ACTION FlowInit:
IF NOT station.xIniting THEN
  station.iStepInit:=0;    
ELSE
//--------------------------------------------初始化步序----------------------------------
CASE station.iStepInit OF	
 0://  
  	IF station.xIniting THEN	
  	  station.iStepInit:=10;	
  	END_IF	
10://复位数据
  station.iStepInit:=20;	
20://停止皮带线
		ATV12.xIMotorStop:=TRUE;
		 station.iStepInit:=999;	
999://初始化完成	
	station.iStepInit:=0;
	station.xInitDone:=TRUE;  
END_CASE
END_IF
END_ACTION

ACTION General:
{region "停止"}
tStopDelay(IN:= fbMachine[1].xManualMode, PT:=T#60S , Q=> , ET=> );
IF tStopDelay.Q THEN
		station.xRunningOffProhibit:=FALSE;
ELSIF  station.iStepAuto =10 THEN
		station.xRunningOffProhibit:=TRUE;
END_IF	 
{endregion}
END_ACTION

ACTION ILC:

//---------------------------------------------------工站可执行-------------------------------------------------------
station.xCanRun :=TRUE ;

//---------------------------------------------------气缸动作条件-------------------------------------------

//变频器
ATV12.xIDeviceRunning:=station.xSingleRunning;
END_ACTION

ACTION Z_Output:

END_ACTION

END_PROGRAM

// ---- POUs/003_FB/0006_ATV/FB_ATV12.TcPOU
FUNCTION_BLOCK FB_ATV12
(*
********************************************************************************
* Name: FB_Encoder
*
* Author:  AutomanH
* Version: 1.0.0
*
* Description:
*   Schneider ATV12 
* Remarks:
*
* Revisions:
* 
*********************************************************************************)
VAR_INPUT
 xIMotorStart:BOOL; //电机启动
 xIMotorStartHMI:BOOL;
 xIMotorStop:BOOL; //电机停止
 xIMotorStopHMI:BOOL;
 xIAutoMode:BOOL;
 xIManualMode:BOOL;
 xIEStop:BOOL;
 xIDeviceRunning:BOOL;
END_VAR
VAR_OUTPUT
 xQMotorStart:BOOL;//变频器电机启动
 arxQMotorSpeedCmd:ARRAY[1..2] OF BOOL;//预制速度
 xQRev:BOOL;//备用
END_VAR
VAR
 	MotorStartR_TRIG:R_TRIG;
	MotorStopR_TRIG:R_TRIG;
	MotorEStopR_TRIG:R_TRIG;
END_VAR

//变频器（2线 漏型）
MotorStartR_TRIG(CLK:=( xIManualMode AND   xIMotorStartHMI ) OR ( (xIAutoMode OR xIDeviceRunning ) AND   xIMotorStart) , Q=> );
MotorStopR_TRIG(CLK:= ( xIManualMode AND   xIMotorStopHMI ) OR ((xIAutoMode OR xIDeviceRunning ) AND xIMotorStop), Q=> );
MotorEStopR_TRIG(CLK:=xIEStop, Q=> );
IF  MotorStartR_TRIG.Q THEN
			xQMotorStart	:=TRUE;//	热缩封膜出料线体¶电机正转/停止
ELSIF	MotorStopR_TRIG.Q	 THEN
			xQMotorStart	:=FALSE;//	热缩封膜出料线体¶电机正转/停止
		
END_IF
	arxQMotorSpeedCmd[1]	:=FALSE;//	热缩封膜出料线体¶电机（预约速度20HZ)
	arxQMotorSpeedCmd[2]	:=TRUE;//	热缩封膜出料线体¶电机（预约速度50HZ）
	
	
	xQRev	:=FALSE;//	热缩封膜出料线体¶电机（未使用）
	
		xIMotorStopHMI:=FALSE;
		xIMotorStop:=FALSE;
		xIMotorStartHMI:=FALSE;
		xIMotorStart:=FALSE;

END_FUNCTION_BLOCK

// ---- POUs/001_Station/S13_Labeling.TcPOU
PROGRAM S13_Labeling
VAR
	//工站
	station					: REFERENCE TO FB_Station:=fbstation[13];
	//气缸
	fbHOZCyl_1			:REFERENCE TO FB_Cylinder:=fbCylinder[36];	//	分料气缸1
	//延时
	arTonDelay :ARRAY[1..20] OF TON;
	//返回值
	UdiReturnValue :ARRAY[1..20] OF UDINT;
	//贴标机
	xLabelJobRdySignal:BOOL;//	贴标机JOBRDY信号
	xLabelReadySignal:BOOL;//	贴标机READY信号
	xLabelErrorSignal:BOOL;//	贴标机ERROR信号
	i: INT;
	xQLabelStart: BOOL;			//	贴标机Start 
	xQLabelRibwarn: BOOL; //	贴标机RIBWARN
	xQLabelReset: BOOL;   //	贴标机RESET  
	
	xQLabelCompleted:BOOL;//贴标完成信号  给PC
	// 贴标到位传感器
	arSensorReached: ARRAY[1..2]of BOOL;
	
	// 设备停止延时
	tStopDelay: TON;
END_VAR

A_Input();
Alarm();
Delay();
FlowAuto();
FlowInit();
General();
ILC();
TipAuto();
TipManual();
Z_Output();

ACTION A_Input:
//气缸
fbHOZCyl_1.xWP_Sensor:=	IxS11HOZCylWP	;//	贴标处推料气缸¶动点
fbHOZCyl_1.xHP_Sensor:=	IxS11HOZCylHP	;//	贴标处推料气缸¶原点
//贴标机

xLabelJobRdySignal:=IxLabelJobRdySignal	;//	贴标机JOBRDY信号
xLabelReadySignal:=IxLabelReadySignal	;//	贴标机READY信号
xLabelErrorSignal:= NOT IxLabelErrorSignal	;//	贴标机ERROR信号

//贴标机到位传感器
arSensorReached[1]:=IxS11SensorReached1	;//	贴标工位¶检查到位传感器1
arSensorReached[2]:=IxS11SensorReached2;//	贴标工位¶检查到位传感器2
END_ACTION

ACTION Alarm:

station.adwAlarm[1].00:=station.xInitTimeout;	  			//S08Label 初始化超时
END_ACTION

ACTION Delay:
(*arTonDelay[01](IN:= , PT:=T#0.1S , Q=> , ET=> );*)//TipAuto使用
arTonDelay[02](IN:= station.iStepAuto=100 , PT:=T#1S , Q=> , ET=> );//贴标识用
arTonDelay[03](IN:=station.iStepAuto =40  , PT:=stData.TimeS[1] , Q=> , ET=> );//计算贴标延时
arTonDelay[04](IN:= , PT:=T#0.1S , Q=> , ET=> );
arTonDelay[05](IN:= , PT:=T#0.1S , Q=> , ET=> );
arTonDelay[06](IN:= , PT:=T#0.1S , Q=> , ET=> );
arTonDelay[07](IN:= , PT:=T#0.1S , Q=> , ET=> );
arTonDelay[08](IN:= , PT:=T#0.1S , Q=> , ET=> );
arTonDelay[09](IN:= , PT:=T#0.1S , Q=> , ET=> );
END_ACTION

ACTION FlowAuto:

//-----------------------------------------初始化是否完成判断----------------------------------------------
IF NOT station.xInitDone 
THEN
 	station.iStepAuto:=0;
 	station.xDone:=FALSE;
ELSIF station.xRunning  OR   station.xRunningOffProhibit
THEN
//-----------------------------------------动作步骤--------------------------------------------------------
CASE station.iStepAuto OF	  
	0: //----Home Step，等待启动----
		IF station.xDisabled 
			AND station.xCanRun 
			AND NOT fbMachine[1].xStopped 
			AND NOT station.xSingleRunning 
		THEN
			station.xDone:=TRUE;
		END_IF
		
		IF  station.xSingleRunning 
			OR station.xCanRun 
			AND NOT station.xDone 
			AND NOT station.xDisabled 
			AND NOT fbMachine[1].xStopped
		THEN
			station.xCycleEnable:=TRUE;
			station.xDone:= FALSE;  
			station.xRunningOffProhibit := TRUE ;//运行中信号Off禁止
			station.iStepAuto:= 10;
		END_IF
    10: //复位数据 
			xQLabelStart:=FALSE;			//	贴标机Start
			station.iStepAuto:=20;
		20://等待第一个传感器感应到
			IF  arSensorReached[1] THEN
						station.iStepAuto:=30;	
			END_IF
		30://等待两个传感器都感应到
				IF  arSensorReached[1]  AND arSensorReached[2] THEN
						station.iStepAuto:=40;	
			END_IF
		40://计算延时触发贴标
				IF   arTonDelay[03].Q THEN
					station.iStepAuto:=100;
				END_IF
		100://开始触发贴标
					xQLabelStart:=TRUE;			//	贴标机Start
					IF	arTonDelay[02].Q THEN
							station.iStepAuto:=110;
					END_IF							
		110://等待贴标完成
					xQLabelStart:=FALSE;			//	贴标机stop
					station.iStepAuto:=999;

		999://----Single Run Finish----
				station.iStepAuto :=0;
				IF NOT station.xSingleContinuousRun THEN
					station.xSingleRunFlag:=FALSE;
				END_IF
				
				station.xCycleEnable:=FALSE;	
				//station.xDone:=TRUE;
			//	station.xRunningOffProhibit := FALSE ;//运行中信号Off禁止
	ELSE
		;	
END_CASE



END_IF
END_ACTION

ACTION FlowInit:
IF NOT station.xIniting THEN
  station.iStepInit:=0;    
ELSE
//--------------------------------------------初始化步序----------------------------------
CASE station.iStepInit OF	
 0://  
  	IF station.xIniting THEN	
  	  station.iStepInit:=10;	
  	END_IF	
10://复位数据
    station.iStepInit:=999;	
		xQLabelStart:=FALSE;			//	贴标机Start
999://初始化完成	
	station.iStepInit:=0;
	station.xInitDone:=TRUE;  
END_CASE
END_IF
END_ACTION

ACTION General:
{region "停止"}
tStopDelay(IN:= fbMachine[1].xManualMode, PT:=T#60S , Q=> , ET=> );
IF tStopDelay.Q THEN
		station.xRunningOffProhibit:=FALSE;
ELSIF  station.iStepAuto =10 THEN
		station.xRunningOffProhibit:=TRUE;
END_IF	 
{endregion}
END_ACTION

ACTION ILC:

//---------------------------------------------------工站可执行-------------------------------------------------------
station.xCanRun :=TRUE ;

//---------------------------------------------------气缸动作条件-------------------------------------------
fbHOZCyl_1.xOffILC	:=	TRUE	;
fbHOZCyl_1.xOnILC	:=	TRUE; 


//---------------------------------------------------伺服动作条件-------------------------------------------
END_ACTION

ACTION TipAuto:

//------------------------------------------------AutoTip Cylinder--------------------------------

//------------------------------------------------AutoTip Servo--------------------------------
//**************************************
END_ACTION

ACTION TipManual:
//--------------------------------------------ManualTip------------------------------------------------------

//-------------------------------------------气缸提示---------------------------------------------------------




/////////////////////////////////////////////////////////////////////////////////////////////////////////////////
END_ACTION

ACTION Z_Output:
(**************************气缸输出********************************)
QxS11HOZCylWP	:=fbHOZCyl_1.xWP_Valve;//	贴标处推料气缸¶动点
QxS11HOZCylHP	:=fbHOZCyl_1.xHP_Valve;//	贴标处推料气缸¶原点
//贴标机
QxLabelStart	:=xQLabelStart;			//	贴标机Start
QxLabelRibwarn:=xQLabelRibwarn;	//	贴标机RIBWARN
QxLabelReset	:=xQLabelReset;		//	贴标机RESET
END_ACTION

END_PROGRAM

// ---- POUs/001_Station/S14_LabelChecking.TcPOU
PROGRAM S14_LabelChecking
VAR
	//工站
	station					: REFERENCE TO FB_Station:=fbstation[14];
	
//气缸
	fbHOZCyl_1			:REFERENCE TO FB_Cylinder:=fbCylinder[37];	//	推料气缸1
	fbHOZCyl_2			:REFERENCE TO FB_Cylinder:=fbCylinder[38];	//	推料气缸2
//相机
	Camera   : 	 REFERENCE TO FB_Camera:=fbCamera[18]; 
	
	//延时
	arTonDelay :ARRAY[1..20] OF TON;
	//返回值
	UdiReturnValue :ARRAY[1..20] OF UDINT;
	i: INT;
 //传感器
	arxBoxCheckSensor: ARRAY[1..2] OF BOOL;
	// //需要推到NG位置
	xNGFlag: BOOL;
	//运行结束
	XFlowAutoDone:BOOL;
		// 设备停止延时
	tStopDelay: TON;
END_VAR

A_Input();
Alarm();
Delay();
FlowAuto();
FlowInit();
General();
ILC();
TipAuto();
TipManual();
Z_Output();

ACTION A_Input:
//气缸
fbHOZCyl_1.xWP_Sensor:=					IxS12HOZCyl_1WP;//	贴标检测工位¶推料气缸1¶动点
fbHOZCyl_1.xHP_Sensor:=					IxS12HOZCyl_1HP;//	贴标检测工位¶推料气缸1¶原点
fbHOZCyl_2.xWP_Sensor:=					IxS12HOZCyl_2HP;//	贴标检测工位¶推料气缸2¶动点
fbHOZCyl_2.xHP_Sensor:=					IxS12HOZCyl_2WP;//	贴标检测工位W推料气缸2¶原点

//传感器
arxBoxCheckSensor[1] :=IxS12SensorReached;	//相机检测处
END_ACTION

ACTION Alarm:
//
station.adwAlarm[1].00:=station.xInitTimeout;	  			//S08Label 初始化超时
//station.adwAlarm[1].01:=TRUE;	  			//S14贴标工位相机检测超时，请检查
END_ACTION

ACTION Delay:
(*arTonDelay[01](IN:= , PT:=T#0.1S , Q=> , ET=> );*)//TipAuto使用
arTonDelay[02](IN:= 	station.iStepAuto=60 , PT:=T#1S , Q=> , ET=> );//已使用
arTonDelay[03](IN:=   , PT:=T#1S , Q=> , ET=> );
arTonDelay[04](IN:= , PT:=T#0.1S , Q=> , ET=> );
arTonDelay[05](IN:= , PT:=T#0.1S , Q=> , ET=> );
arTonDelay[06](IN:= , PT:=T#0.1S , Q=> , ET=> );
arTonDelay[07](IN:= , PT:=T#0.1S , Q=> , ET=> );
arTonDelay[08](IN:= , PT:=T#0.1S , Q=> , ET=> );
arTonDelay[09](IN:= , PT:=T#0.1S , Q=> , ET=> );
END_ACTION

ACTION FlowAuto:

//-----------------------------------------初始化是否完成判断----------------------------------------------
IF NOT station.xInitDone 
THEN
 	station.iStepAuto:=0;
 	station.xDone:=FALSE;
ELSIF station.xRunning  OR   station.xRunningOffProhibit
THEN
//-----------------------------------------动作步骤--------------------------------------------------------
CASE station.iStepAuto OF	  
	0: //----Home Step，等待启动----
		IF station.xDisabled 
			AND station.xCanRun 
			AND NOT fbMachine[1].xStopped 
			AND NOT station.xSingleRunning 
		THEN
			station.xDone:=TRUE;
		END_IF
		
		IF  station.xSingleRunning 
			OR station.xCanRun 
			AND NOT station.xDone 
			AND NOT station.xDisabled 
			AND NOT fbMachine[1].xStopped
		THEN
			station.xCycleEnable:=TRUE;
			station.xDone:= FALSE;  
			station.xRunningOffProhibit := TRUE ;//运行中信号Off禁止
			station.iStepAuto:= 10;
		END_IF
  10: //复位数据 
			xFlowAutoDone:=FALSE;	
			xNGFlag:=FALSE;
			sCamera_TO_Plc.iS13Result[1]:=0;
			station.iStepAuto:=20;
	20://等待传感器检测
			IF  arxBoxCheckSensor[1]  THEN
					station.iStepAuto:=30;
			END_IF
	30://水平阻挡气缸伸出
				fbHOZCyl_1.xAuto:=TRUE;
			IF	fbHOZCyl_1.xWP_Delay THEN
			 	station.iStepAuto:=40;
			END_IF
	40://阻挡气缸下降
			fbHOZCyl_2.xAuto:=FALSE;
			IF	fbHOZCyl_2.xHP_Delay THEN
			 	station.iStepAuto:=50;
			END_IF
	50://收回水平阻挡气缸
				fbHOZCyl_1.xAuto:=FALSE;
			IF	fbHOZCyl_1.xHP_Delay THEN
			 	station.iStepAuto:=60;
			END_IF
	60://等待
				IF   arTonDelay[02].Q THEN
							station.iStepAuto:=70;
				END_IF
	70://相机检测
				Camera.xlTrigger:=TRUE;
					station.iStepAuto:=75;
	75://等待相机响应
			IF    Camera.xQBusy THEN
				station.iStepAuto:=80;	
			END_IF
	80://等待相机完成
			 IF   Camera.xQDone THEN
				 station.iStepAuto:=90;	
			 ELSIF Camera.xQAlarm THEN
					Camera.xlInit:=TRUE;
					station.iStepAuto:=70;
					station.adwAlarm[1].01:=TRUE;	//S14贴标工位相机检测超时，请检查	
			 END_IF
	90://处理相机结果
			IF 	sCamera_TO_Plc.iS13Result[1] =1  THEN
				//相机拍照结果， 1=OK 2=NG，触发前PLC清除	
					xNGFlag:=FALSE;
					station.iStepAuto:=100;
			ELSIF sCamera_TO_Plc.iS13Result[1] =2 THEN
			 		xNGFlag:=TRUE;
			 		station.iStepAuto:=100;
			END_IF
	100://阻挡气缸抬起
			fbHOZCyl_2.xAuto:=TRUE;
			IF	fbHOZCyl_2.xWP_Delay THEN
			 	station.iStepAuto:=110;
			END_IF
	110://等待传感器
			IF  NOT  arxBoxCheckSensor[1] THEN
			 		station.iStepAuto:=999;
			END_IF
	
	999://----Single Run Finish----
		xFlowAutoDone:=TRUE;	
		station.iStepAuto :=0;
		IF NOT station.xSingleContinuousRun THEN
			station.xSingleRunFlag:=FALSE;
		END_IF
		
		station.xCycleEnable:=FALSE;	
	//	station.xDone:=TRUE;
	//	station.xRunningOffProhibit := FALSE ;//运行中信号Off禁止
	ELSE
		;	
END_CASE



END_IF
END_ACTION

ACTION FlowInit:
IF NOT station.xIniting THEN
  station.iStepInit:=0;    
ELSE
//--------------------------------------------初始化步序----------------------------------
CASE station.iStepInit OF	
 0://  
  	IF station.xIniting THEN	
  	  station.iStepInit:=10;	
  	END_IF	
10://复位数据
    station.iStepInit:=20;	
20://阻挡气缸回原
			fbHOZCyl_1.xInit:=TRUE;
		IF  fbHOZCyl_1.xHP_Delay   THEN
				station.iStepInit:=30;	
		END_IF
30://升降气缸回原
			fbHOZCyl_2.xInit:=TRUE;
		IF  fbHOZCyl_2.xHP_Delay   THEN
				station.iStepInit:=999;	
		END_IF
999://初始化完成	
	station.iStepInit:=0;
	station.xInitDone:=TRUE;  
END_CASE
END_IF
END_ACTION

ACTION General:
{region "停止"}
tStopDelay(IN:= fbMachine[1].xManualMode, PT:=T#60S , Q=> , ET=> );
IF tStopDelay.Q THEN
		station.xRunningOffProhibit:=FALSE;
ELSIF  station.iStepAuto =10 THEN
		station.xRunningOffProhibit:=TRUE;
END_IF	 
{endregion}
END_ACTION

ACTION ILC:

//---------------------------------------------------工站可执行-------------------------------------------------------
station.xCanRun :=TRUE ;

//---------------------------------------------------气缸动作条件-------------------------------------------
fbHOZCyl_1.xOffILC	:=	TRUE	;
fbHOZCyl_1.xOnILC	:=	TRUE; 

fbHOZCyl_2.xOffILC	:=	TRUE	;
fbHOZCyl_2.xOnILC	:=	TRUE; 


//---------------------------------------------------伺服动作条件-------------------------------------------

Camera.xIDeviceRunning:=TRUE;
END_ACTION

ACTION TipAuto:

//------------------------------------------------AutoTip Cylinder--------------------------------
	
//------------------------------------------------AutoTip Servo--------------------------------
//**************************************
END_ACTION

ACTION TipManual:
//--------------------------------------------ManualTip------------------------------------------------------

//-------------------------------------------气缸提示---------------------------------------------------------




/////////////////////////////////////////////////////////////////////////////////////////////////////////////////
END_ACTION

ACTION Z_Output:
(**************************气缸输出********************************)
QxS12HOZCyl_1WP	:=fbHOZCyl_1.xWP_Valve;//	贴标检测工位¶推料气缸1¶动点
QxS12HOZCyl_1HP	:=fbHOZCyl_1.xHP_Valve;//	贴标检测工位¶推料气缸1¶原点
QxS12HOZCyl_2WP	:=fbHOZCyl_2.xWP_Valve;//	贴标检测工位¶推料气缸2¶动点
QxS12HOZCyl_2HP	:=fbHOZCyl_2.xHP_Valve;//	贴标检测工位¶推料气缸2¶原点
END_ACTION

END_PROGRAM

// ---- POUs/001_Station/S15_NG.TcPOU
PROGRAM S15_NG
VAR
	//工站
	station					: REFERENCE TO FB_Station:=fbstation[15];
	//气缸
	fbHOZCyl_1			:REFERENCE TO FB_Cylinder:=fbCylinder[39];	//	分料气缸1
	fbHOZCyl_2			:REFERENCE TO FB_Cylinder:=fbCylinder[40];	//	分料气缸2
	
	
	//延时
	arTonDelay :ARRAY[1..20] OF TON;
	//返回值
	UdiReturnValue :ARRAY[1..20] OF UDINT;
	i: INT;
	NGFlagR_TRIG: R_TRIG;
	// Box检测到位
	arxBoxCheckSensor: ARRAY[1..2] of BOOL;
	// //相机检测NG信号
	xNGFlag: BOOL;
			// 设备停止延时
	tStopDelay: TON;
END_VAR

A_Input();
Alarm();
Delay();
FlowAuto();
FlowInit();
General();
ILC();
TipAuto();
TipManual();
Z_Output();

ACTION A_Input:
//气缸
fbHOZCyl_1.xWP_Sensor:=IxS13HOZCyl_1WP	;//	NG推料气缸1¶动点
fbHOZCyl_1.xHP_Sensor:=IxS13HOZCyl_1HP	;//	NG推料气缸1¶原点
fbHOZCyl_2.xWP_Sensor:=IxS13HOZCyl_2WP	;//	NG推料气缸2¶动点
fbHOZCyl_2.xHP_Sensor:=IxS13HOZCyl_2HP	;//	NG推料气缸2¶原点
//退料检测
arxBoxCheckSensor[1] :=IxS13SensorReached1; //NG推料处检测
arxBoxCheckSensor[2] :=IxS13SensorReached2; //NG流道处检测
END_ACTION

ACTION Alarm:
//
station.adwAlarm[1].00:=station.xInitTimeout;	  			//S08Label 初始化超时
END_ACTION

ACTION Delay:
(*arTonDelay[01](IN:= , PT:=T#0.1S , Q=> , ET=> );*)//TipAuto使用
arTonDelay[02](IN:=  , PT:=T#1S , Q=> , ET=> );
arTonDelay[03](IN:=   , PT:=T#1S , Q=> , ET=> );
arTonDelay[04](IN:= , PT:=T#0.1S , Q=> , ET=> );
arTonDelay[05](IN:= , PT:=T#0.1S , Q=> , ET=> );
arTonDelay[06](IN:= , PT:=T#0.1S , Q=> , ET=> );
arTonDelay[07](IN:= , PT:=T#0.1S , Q=> , ET=> );
arTonDelay[08](IN:= , PT:=T#0.1S , Q=> , ET=> );
arTonDelay[09](IN:= , PT:=T#0.1S , Q=> , ET=> );
END_ACTION

ACTION FlowAuto:

//-----------------------------------------初始化是否完成判断----------------------------------------------
IF NOT station.xInitDone 
THEN
 	station.iStepAuto:=0;
 	station.xDone:=FALSE;
ELSIF station.xRunning  OR   station.xRunningOffProhibit
THEN
//-----------------------------------------动作步骤--------------------------------------------------------
CASE station.iStepAuto OF	  
	0: //----Home Step，等待启动----
		IF station.xDisabled 
			AND station.xCanRun 
			AND NOT fbMachine[1].xStopped 
			AND NOT station.xSingleRunning 
		THEN
			station.xDone:=TRUE;
		END_IF
		
		IF  station.xSingleRunning 
			OR station.xCanRun 
			AND NOT station.xDone 
			AND NOT station.xDisabled 
			AND NOT fbMachine[1].xStopped
		THEN
			station.xCycleEnable:=TRUE;
			station.xDone:= FALSE;  
			station.xRunningOffProhibit := TRUE ;//运行中信号Off禁止
			station.iStepAuto:= 10;
		END_IF
    10: //复位数据 
			station.iStepAuto:=20;
		20://等待NG信号
			IF  xNGFlag THEN
			 			station.iStepAuto:=30;
			ELSE
			 		station.iStepAuto:=999;
			END_IF
		30://等待到位信号
			IF  arxBoxCheckSensor[1] THEN
				 station.iStepAuto:=40;
			END_IF
		40://水平推料气缸伸出
			fbHOZCyl_1.xAuto:=TRUE;
			IF fbHOZCyl_1.xWP_Delay THEN
			 	 station.iStepAuto:=50;
			END_IF
		50://水平退料气缸收回
				fbHOZCyl_1.xAuto:=FALSE;
			IF fbHOZCyl_1.xHP_Delay THEN
			 	 station.iStepAuto:=60;
			END_IF
		60://等待NG流道检测
			//IF  arxBoxCheckSensor[2] THEN
			 	 station.iStepAuto:=70;
			//END_IF
		70://NG流道退料气缸伸出
			fbHOZCyl_2.xAuto:=TRUE;
			IF fbHOZCyl_2.xWP_Delay THEN
			 	 station.iStepAuto:=80;
			END_IF
		80://NG流道退料气缸收回
			fbHOZCyl_2.xAuto:=FALSE;
			IF fbHOZCyl_2.xHP_Delay THEN
			 	 station.iStepAuto:=90;
			END_IF
		90://检查NG物料
			IF NOT  arxBoxCheckSensor[2] THEN
			 	 station.iStepAuto:=999;
			END_IF
	999://----Single Run Finish----
			xNGFlag:=FALSE;	
			station.iStepAuto :=0;
			IF NOT station.xSingleContinuousRun THEN
				station.xSingleRunFlag:=FALSE;
			END_IF
			
			station.xCycleEnable:=FALSE;	
		//	station.xDone:=TRUE;
		//	station.xRunningOffProhibit := FALSE ;//运行中信号Off禁止
	ELSE
		;	
END_CASE



END_IF
END_ACTION

ACTION FlowInit:
IF NOT station.xIniting THEN
  station.iStepInit:=0;    
ELSE
//--------------------------------------------初始化步序----------------------------------
CASE station.iStepInit OF	
 0://  
  	IF station.xIniting THEN	
  	  station.iStepInit:=10;	
  	END_IF	
10://复位数据
    station.iStepInit:=20;
20://气缸回原
		fbHOZCyl_1.xInit:=TRUE;
		fbHOZCyl_2.xInit:=TRUE;	
	IF  fbHOZCyl_1.xHP_Delay AND
		 fbHOZCyl_2.xHP_Delay THEN
		 station.iStepInit:=999;
	END_IF
999://初始化完成	
	station.iStepInit:=0;
	station.xInitDone:=TRUE;  
END_CASE
END_IF
END_ACTION

ACTION General:
{region '相机检测出NG的信号传递'}
NGFlagR_TRIG(CLK:= S14_LabelChecking.xFlowAutoDone AND S14_LabelChecking.xNGFlag, Q=> );
IF  NGFlagR_TRIG.Q THEN
		xNGFlag:=TRUE;		
END_IF
	 
{endregion}

{region "停止"}
tStopDelay(IN:= fbMachine[1].xManualMode, PT:=T#60S , Q=> , ET=> );
IF tStopDelay.Q THEN
		station.xRunningOffProhibit:=FALSE;
ELSIF  station.iStepAuto =10 THEN
		station.xRunningOffProhibit:=TRUE;
END_IF	 
{endregion}
END_ACTION

ACTION ILC:

//---------------------------------------------------工站可执行-------------------------------------------------------
station.xCanRun :=TRUE ;

//---------------------------------------------------气缸动作条件-------------------------------------------
fbHOZCyl_1.xOffILC	:=	TRUE;
fbHOZCyl_1.xOnILC	:=	fbHOZCyl_2.xHP_Sensor; 

fbHOZCyl_2.xOffILC	:=	TRUE	;
fbHOZCyl_2.xOnILC	:=	TRUE; 

//---------------------------------------------------伺服动作条件-------------------------------------------
END_ACTION

ACTION TipAuto:

//------------------------------------------------AutoTip Cylinder--------------------------------

//------------------------------------------------AutoTip Servo--------------------------------
//**************************************
END_ACTION

ACTION TipManual:
//--------------------------------------------ManualTip------------------------------------------------------

//-------------------------------------------气缸提示---------------------------------------------------------




/////////////////////////////////////////////////////////////////////////////////////////////////////////////////
END_ACTION

ACTION Z_Output:
(**************************气缸输出********************************)
QxS13HOZCyl_1WP	:=fbHOZCyl_1.xWP_Valve;//	NG推料气缸1¶动点
QxS13HOZCyl_1HP	:=fbHOZCyl_1.xHP_Valve;//	NG推料气缸1¶原点
QxS13HOZCyl_2WP	:=fbHOZCyl_2.xWP_Valve;//	NG推料气缸2¶动点
QxS13HOZCyl_2HP	:=fbHOZCyl_2.xHP_Valve;//	NG推料气缸2¶原点
END_ACTION

END_PROGRAM

// ---- POUs/001_Station/S16_Unloading.TcPOU
PROGRAM S16_Unloading
VAR
 //工站
	station					: REFERENCE TO FB_Station:=fbstation[16];
END_VAR

FlowAuto();
FlowInit();
ILC();

ACTION FlowAuto:

//-----------------------------------------初始化是否完成判断----------------------------------------------
IF NOT station.xInitDone 
THEN
 	station.iStepAuto:=0;
 	station.xDone:=FALSE;
ELSIF station.xRunning  
THEN
//-----------------------------------------动作步骤--------------------------------------------------------
CASE station.iStepAuto OF	  
	0: //----Home Step，等待启动----
		IF station.xDisabled 
			AND station.xCanRun 
			AND NOT fbMachine[1].xStopped 
			AND NOT station.xSingleRunning 
		THEN
			station.xDone:=TRUE;
		END_IF
		
		IF  station.xSingleRunning 
			OR station.xCanRun 
			//AND NOT station.xDone 
			AND NOT station.xDisabled 
			AND NOT fbMachine[1].xStopped
		THEN
			station.xCycleEnable:=TRUE;
			//station.xDone:= FALSE;  
			
			station.iStepAuto:= 10;
		END_IF
    10: //复位数据 
			station.iStepAuto :=999;
		
	999://----Single Run Finish----
			
		station.iStepAuto :=0;
		IF NOT station.xSingleContinuousRun THEN
			station.xSingleRunFlag:=FALSE;
		END_IF
		
		station.xCycleEnable:=FALSE;	
		(*station.xDone:=TRUE;*)
	ELSE
		;	
END_CASE
END_IF
END_ACTION

ACTION FlowInit:
IF NOT station.xIniting THEN
  station.iStepInit:=0;    
ELSE
//--------------------------------------------初始化步序----------------------------------
CASE station.iStepInit OF	
 0://  
  	IF station.xIniting THEN	
  	  station.iStepInit:=10;	
  	END_IF	
10://复位数据
	station.iStepInit:=999;
999://初始化完成	
	station.iStepInit:=0;
	station.xInitDone:=TRUE;  
END_CASE
END_IF
END_ACTION

ACTION ILC:

//---------------------------------------------------工站可执行-------------------------------------------------------
station.xCanRun :=TRUE ;

//---------------------------------------------------气缸动作条件-------------------------------------------
END_ACTION

END_PROGRAM

// ---- POUs/002_Machine/ControlMachine.TcPOU
PROGRAM ControlMachine
VAR_input
	xAlarm                      	: BOOL;
	tonEmptyDone	: TON;					//Empty Done Delay
	bEmptyDone                  	: BOOL ;
	
	
END_VAR
VAR
	i,j : INT ;
	_xMaterialOnFlag : BOOL ;//环形线
	MachineLampR_TRIG:R_TRIG;
	MachineLampF_TRIG:F_TRIG;
	
	tTimeoutAlarm: TON;
	tCounterR_TRIG: R_TRIG;
	tCounter1R_TRIG: R_TRIG;
	tCounter2R_TRIG: R_TRIG;
	tPCAlarmR_TRIG: R_TRIG;
	artEmptyMachineR_TRIG:ARRAY[1..2] OF R_TRIG;
END_VAR

A_Input();
Safety();
Waiting();
Timeout();
Alarm();
CycleTime();
Tip();
InitDone();
EmptyDone();
General();
Z_Output();

ACTION A_Input:
FOR i:=1 TO gc_uiAxisNum BY 1 DO
	arAxisSensorP[i]:=arAxisSensor[i].0;
	arAxisSensorN[i]:=arAxisSensor[i].1;
	arAxisSensorH[i]:=arAxisSensor[i].2;
END_FOR
END_ACTION

ACTION Alarm:
//----机台状态提示---//
fbMachine[1].dwMessage[1].00			:=	fbMachine[1].xRunning;			//设备自动中
fbMachine[1].dwMessage[1].01		    :=	fbMachine[1].xStopped;			//设备停止状态
fbMachine[1].dwMessage[1].02			:=	fbMachine[1].xPaused;			//设备暂停状态
fbMachine[1].dwMessage[1].03			:=	fbMachine[1].xAlarm;			//设备报警中
fbMachine[1].dwMessage[1].04			:=	fbMachine[1].xIniting;			//设备初始化中
fbMachine[1].dwMessage[1].05			:=	fbMachine[1].xEmptying;			//设备清料中

//----机台报警信息----
//IF NOT  fbMachine[1].xAirOn THEN
//	fbMachine[1].dwAlarm[1].00:=TRUE; //[M01.00] 设备气压报警
//	;
//END_IF

//急停被按下
IF NOT IxSafetyRelayOK THEN 
	fbMachine[1].dwAlarm[1].03:=TRUE; //[M01.03] 设备急停被按下
END_IF
IF   sModbus_200SMART.iStatus =3 THEN 
 		fbMachine[1].dwAlarm[1].04:=TRUE; //[M01.04] 热缩封膜机急停被按下
END_IF
//心跳
	IF  fbAlive[1].xQAliveError THEN
		fbMachine[1].dwAlarm[1].05:=TRUE; //[M01.05] 未检测到相机心跳1
	END_IF
	IF  fbAlive[2].xQAliveError THEN
		fbMachine[1].dwAlarm[1].06:=TRUE; //[M01.06] 未检测到相机心跳2
	END_IF
	IF  fbAlive[3].xQAliveError THEN
		fbMachine[1].dwAlarm[1].07:=TRUE; //[M01.07] 未检测到相机心跳3
	END_IF
//IF  fbAlive[4].xQAliveError THEN
//	fbMachine[1].dwAlarm[1].08:=TRUE; //[M01.08] 未检测到工控机1心跳
//END_IF
///	IF  fbAlive[5].xQAliveError THEN
//		fbMachine[1].dwAlarm[1].09:=TRUE; //[M01.09] 未检测到工控机2心跳
//	END_IF
//	IF  fbAlive[6].xQAliveError THEN
//		fbMachine[1].dwAlarm[1].10:=TRUE; //[M01.10] 未检测到工控机3心跳
//	END_IF
	IF  fbAlive[7].xQAliveError THEN
		fbMachine[1].dwAlarm[1].11:=TRUE; //[M01.11] 未检测到热缩封膜机心跳
	END_IF
////模块状态
	IF  fbEhterCATSlaveMonitor[1].xQError THEN
		fbMachine[1].dwAlarm[1].12:=TRUE; //[M01.05] ET01电柜EtherCAT总线报错
	END_IF
	IF  fbEhterCATSlaveMonitor[2].xQError THEN
		fbMachine[1].dwAlarm[1].13:=TRUE; //[M01.05] ET02电柜EtherCAT总线报错
	END_IF
	IF  fbEhterCATSlaveMonitor[3].xQError THEN
		fbMachine[1].dwAlarm[1].14:=TRUE; //[M01.05] ET03电柜EtherCAT总线报错
	END_IF
	IF  fbEhterCATSlaveMonitor[4].xQError THEN
		fbMachine[1].dwAlarm[1].15:=TRUE; //[M01.05] ET04电柜EtherCAT总线报错
	END_IF

	fbMachine[1].dwAlarm[1].16:=(sPLC_From_PC.iPCAlarm =1); //[M01.16] PC报警
	
	
//----工站报警汇总----

xAlarm:= FALSE;							//先复位
FOR i :=1 TO gc_uiStationNum DO 
  IF fbStation[i].xAlarm THEN		//整机故障单独 
    xAlarm:=TRUE; 
  END_IF
END_FOR

//----机台报警----
fbMachine[1].xAlarm:=
  fbMachine[1].dwAlarm[1]<>0
	OR fbMachine[1].dwAlarm[2]<>0
	OR fbMachine[1].dwAlarm[3]<>0
	OR fbMachine[1].dwAlarm[4]<>0
	OR fbMachine[1].dwAlarm[5]<>0
	OR xAlarm;
END_ACTION

ACTION CycleTime:
//**************************计算循环周期*******************************///
END_ACTION

ACTION EmptyDone:
{region"第一站清料信号"}
artEmptyMachineR_TRIG[1](CLK:=fbMachine[1].xEmptying, Q=> );
IF artEmptyMachineR_TRIG[1].Q THEN
			fbStation[1].xEmptying:=TRUE;
END_IF
{region}
	 
{region "复位各工位的清空完成信号"}
artEmptyMachineR_TRIG[2](CLK:=fbMachine[1].xEmptyDone, Q=> );
IF artEmptyMachineR_TRIG[2].Q THEN
		FOR i:=1 TO gc_uiStationNum BY 1 DO
			fbStation[i].xEmptyDone:=FALSE;
		END_FOR 
END_IF
{endregion}
{region "整机请料完成信号"}
FOR i:=1 TO gc_uiStationNum BY 1 DO
 		IF NOT fbStation[i].xEmptyDone THEN
			EXIT;
		ELSIF i =		gc_uiStationNum THEN
				fbMachine[1].xEmptyDone:=TRUE;
		END_IF
END_FOR
{endregion}
END_ACTION

ACTION General:

//设备总产量
  fbMachine[1].udiTotal := fbMachine[1].udiGoods + fbMachine[1].udiBads ;

//产量清除
  IF fbMachine[1].xClearCountData THEN 
	  fbMachine[1].udiGoods := fbMachine[1].udiBads := 0 ;
	  fbMachine[1].xClearCountData:=FALSE;
  END_IF
  
//产品计数
(*
tCounterR_TRIG(CLK:=S07_Unloading.xBothPartGoodFlag, Q=> );
tCounter1R_TRIG(CLK:=S07_Unloading.xOnePartGoodFlag , Q=> );
tCounter2R_TRIG(CLK:=S07_Unloading.xOnePartBadFlag , Q=> );
*)
IF  tCounterR_TRIG.Q THEN
	fbMachine[1].udiGoods := fbMachine[1].udiGoods + 2;	//设备OK产品计数
ELSIF  tCounter1R_TRIG.Q  THEN
	fbMachine[1].udiGoods := fbMachine[1].udiGoods + 1;	//设备OK产品计数
ELSIF  tCounter2R_TRIG.Q THEN
	fbMachine[1].udiBads := fbMachine[1].udiBads + 1;	//设备OK产品计数	
END_IF
END_ACTION

ACTION InitDone:

//------------------------------------------------初始化完成汇总-------------------------------------

fbMachine[1].xInitDone:=TRUE;//先置位
FOR j :=1 TO gc_uiStationNum DO 
  IF NOT fbStation[j].xInitDone
  THEN 
    fbMachine[1].xInitDone:=FALSE; 
  END_IF
END_FOR
END_ACTION

ACTION Safety:
//-------------------------------------------------安全信号------------------------------------------------------

//fbMachine[1].xDoorClosed:= fbSafetyDoor[1].xLocked ;
						
//fbSafetyDoor[1].xUnlock:= FALSE;
fbMachine[1].xDoorClosed := TRUE ;

fbMachine[1].xEStop :=IxSafetyRelayOK ;					   

fbMachine[1].xKey := TRUE;

fbMachine[1].xAirOn :=  IxAirPressure OR true;

fbMachine[1].xSafety:=fbMachine[1].xDoorClosed 
						AND fbMachine[1].xEStop 
						AND fbMachine[1].xAirOn 
						AND fbMachine[1].xKey  AND   sModbus_200SMART.iStatus <>3;
END_ACTION

ACTION Timeout:

END_ACTION

ACTION Tip:
//------------------------------------------------提示汇总-----------------------------------------------
//----手动提示----
fbMachine[1].xManualTip                :=FALSE;//先复位
FOR j:=1 TO gc_uiStationNum DO 
  IF fbStation[j].xManualTip THEN 
   fbMachine[1].xManualTip            :=TRUE; 
  END_IF
END_FOR

//----自动提示----
fbMachine[1].xAutoTip                  :=FALSE;//先复位
FOR j :=1 TO gc_uiStationNum DO 
  IF fbStation[j].xAutoTip
  THEN 
   fbMachine[1].xAutoTip              :=TRUE; 
  END_IF
END_FOR

fbMachine[1].xTip                      :=(fbMachine[1].xManualTip OR fbMachine[1].xAutoTip);
/////////////////////////////////////////////////////////////////////////////////////////////////////////
END_ACTION

ACTION Waiting:

END_ACTION

ACTION Z_Output:
////设备照明
MachineLampR_TRIG(CLK:= xMachineLamp, Q=> );
MachineLampF_TRIG(CLK:= xMachineLamp, Q=> );
IF  MachineLampR_TRIG.Q THEN
 	QxMachineLamp1Control:=TRUE	;//	日光灯1控制
  QxMachineLamp2Control:=TRUE	;//	日光灯2控制
	QxMachineLamp3Contorl:=TRUE	;//	日光灯控制
ELSIF   MachineLampF_TRIG.Q THEN
  QxMachineLamp1Control:=FALSE	;//	日光灯1控制
  QxMachineLamp2Control:=FALSE	;//	日光灯2控制
	QxMachineLamp3Contorl:=FALSE	;//	日光灯控制
END_IF
END_ACTION

END_PROGRAM

// ---- POUs/002_Machine/CallStandard.TcPOU
PROGRAM CallStandard
VAR_INPUT
	{attribute 'hide'}
	fb_Blinker					: ARRAY[1..10] OF FB_Blinker;//自定义脉冲发生功能块
	bWindowColseHmi             : ARRAY[1..5]OF BOOL ; //窗口关闭
END_VAR

VAR
	xCylinder_First  	: BOOL ;
	xAxis_First 		: BOOL ;
	xAxisHome_First 	: BOOL ;
	xMachine_First 		: BOOL ;
 	xStation_First 		: BOOL ;
    xRGI4_First 		: BOOL ;
	xEPSRobot_First 	: BOOL ;
	xRefrigerator_first : BOOL ;
	_firstFuShiPXF		: BOOL ;
	_firstTURINRobot     :BOOL;
	_xCalFirstCycle		 :BOOL;
	
	
	i: INT;j,k,eps,rgi,l,m,n,iIndex,t,mac,infor,iRec,q : INT ;
	arrayMoveFalse : ARRAY[1..gc_uiAxisMoveNum] OF BOOL ;
    st_RGI_IOData : ST_RGI_14_IOData;
	
	sModeOperation	AT %Q*: ARRAY[1..gc_uiAxisNum] OF SINT;			//操作模式
	controlword AT %Q* : ARRAY[1..gc_uiAxisNum] OF UINT;
	nctrl1 		AT %I* : ARRAY[1..gc_uiAxisNum] OF USINT;
	nctrl2		AT %I*  : ARRAY[1..gc_uiAxisNum] OF USINT;	
	
    
	fbWritePersistentData		: FB_WritePersistentData;//系统自带保存Persistent数据功能块
	
	strDateTime: STRING(10);
	
	stDateTime: DUT_TIMESET;
	
	xRecipeAxisParSetButton : BOOL ;
	xRecipeRGI14ParSetButton : BOOL ;
	StepHistoryR_TRIG	:R_TRIG;
	SFCTrans: BOOL;
	iInfo: INT;
	arRefSwitchCheckSensor:ARRAY[1..gc_uiAxisNum] OF BOOL;
	fbReference_TRIG:ARRAY[1..gc_uiAxisNum] OF R_TRIG;
	
	
	
	StepAutoTransR_TRIG: ARRAY[1..gc_uiStationNum] OF R_TRIG;
	stepInitTransR_TRIG:ARRAY[1..gc_uiStationNum] OF R_TRIG;
	tTonoff1s: TON;
	tTonOn1s: TON;
	rstStartCoordinate: INT;
	bMachine_First: BOOL;
	_FirstCycle: BOOL;
	bAxisHome_First: BOOL;
	A: INT;
	tLamp2R_TRIG: R_TRIG;
	tLamp3R_TRIG: R_TRIG;
	tLampR_TRIG: R_TRIG;
	tLamp1R_TRIG: R_TRIG;
	
	iSlavePort: INT;
	
	xMonitoring: BOOL;
	xReset: BOOL;
	xtest: BOOL;
END_VAR

A_Input();
ACT_Axis();
ACT_AxisHome();
ACT_Cylinder();
ACT_Machine();
ACT_Proface();
ACT_RGI_14();
ACT_Station();
ACT_System();
ACT_WritePersistentData();
ACT_GetTime();
ACT_Comm();
ACT_UPS();
ACT_Recipe();
ACT_Z_ERG_20();
ACT_Camera();
//ACT_PeristalticPump();
//ACT_PeristalticPump_1();
ACT_TURINRobot();
//ACT_MT_MCK();
ACT_MT_MCK_1();
ACT_Alive();
ACT_EtherCATSlaveState();
ACT_FuShiPXF();
ACT_M0dbus_200Smart();
ACT_Encoder();
ACT_ATV12();
ACT_SmcVacuum();
ACT_LoadCell();
ACT_Cimcor();
ACT_EasyPump();
//ACT_ERG_20C();

ACTION A_Input:
IF   fbTURINContorl[1].pSysFromRobot[2].0 THEN
 		xMonitoring:=TRUE;
END_IF
END_ACTION

ACTION ACT_Alive:
//检测心跳
fbAlive[1].iAliveSingle:=sCamera_TO_Plc.iCameraAlive[1];
fbAlive[2].iAliveSingle:=sCamera_TO_Plc.iCameraAlive[2];
fbAlive[3].iAliveSingle:=sCamera_TO_Plc.iCameraAlive[3];
fbAlive[4].iAliveSingle:=sPLC_From_PC.iPCAlive;
fbAlive[7].iAliveSingle:=sModbus_200SMART.iAlive;

//PLC心跳
 IF  fbAlive[5].xQAlive THEN
		sPLC_TO_PC.iPLCALive:=1;
 ELSE
		sPLC_TO_PC.iPLCALive:=0;
 END_IF

FOR i:=1 TO gc_AliveNum DO
		fbAlive[i](iAliveSingle:= , xQAlive=> , xQAliveError=> );
END_FOR
END_ACTION

ACTION ACT_ATV12:
fbATV12(
	xIMotorStart:= , 
	xIMotorStartHMI:= , 
	xIMotorStop:= , 
	xIMotorStopHMI:= , 
	xIEStop:=NOT fbMachine[1].xEStop , 
	xIAutoMode:=	fbMachine[1].xAutoMode , 
	xIManualMode:= fbMachine[1].xManualMode, 
	xIDeviceRunning:= , 
	xQMotorStart=>QxMotorForward, //	热缩封膜出料线体¶电机正转/停止 , 
	arxQMotorSpeedCmd=> , 
	xQRev=>QxMotorStop	);//	热缩封膜出料线体¶电机（未使用） 
	
	QxMotorBackward	:=fbATV12.arxQMotorSpeedCmd[1];//	热缩封膜出料线体¶电机（预约速度20HZ)
	QxMotorReserve	:=fbATV12.arxQMotorSpeedCmd[2];//	热缩封膜出料线体¶电机（预约速度50HZ）
END_ACTION

ACTION ACT_Axis:
//上电复位
IF NOT xAxis_First THEN
  FOR i :=1 TO (gc_uiAxisNum) DO 
      	fbAxis[i].xAlarmResetHmi                   :=     			//HMI_故障复位
	    fbAxis[i].xPowerHmi                        :=     			//HMI_使能
	    fbAxis[i].xJogForwardHmi                   :=     			//HMI_正点
	    fbAxis[i].xJogBackwardsHmi                 :=     			//HMI_反点
	    fbAxis[i].xHomeHmi                         :=     			//HMI_回零
	    fbAxis[i].xStopHmi                         :=FALSE;			//HMI_停止
	    fbAxis[i].xMoveHmi                         :=arrayMoveFalse;			//HMI_P点
  END_FOR                                       			
      xAxis_First                           :=TRUE;
END_IF

FOR j:=1 TO gc_uiAxisNum DO
    fbAxis[j](
	Axis := Axis[j], 
	xEStop:= fbMachine[1].xEStop , 
	xKey:=fbMachine[1].xKey  , 
	xSafety:=fbMachine[1].xSafety   , 
	xManualMode:=fbMachine[1].xManualMode  , 
	xAutoMode:=fbMachine[1].xAutoMode , 
	xAlarmReset:=fbMachine[1].xReset  , 
	rJogAcceleration:=stData.Axis[j].rAcceleration , 
	rJogDeceleration:=stData.Axis[j].rDeceleration , 
	rMoveAcceleration:=stData.Axis[j].rAcceleration , 
	rMoveDeceleration:=stData.Axis[j].rDeceleration , 
	rJogVelocity:=stData.Axis[j].rJogVelocity , 
	rManualVelocity:=stData.Axis[j].rManualVelocity , 
	rAutoVelocity:=stData.Axis[j].rAutoVelocity , 
	rMovePosition:=stData.Axis[j].rMovePosition , 
	rMoveVelocity:=stData.Axis[j].rMoveVelocity , 
	rRelativeDistance:=stData.Axis[j].rRelativeDistance , 
	rRelativeVelocity:=stData.Axis[j].rRelativeVelocity , 
	rVelocityVel:=stData.Axis[j].rVelocityVel , 
	rVelocityAcc:=stData.Axis[j].rAcceleration , 
	rVelocityDec:=stData.Axis[j].rDeceleration , 
	xIRefSwitch:= arAxisSensorH[j], 
	xIResetRefPosCheck:= , 
	xPowerOn=> , 
	xReady=> , 
	xRelativeDone1=> , 
	xError=> , 
	nErrorID=> , 
	rActTorque=> , 
	rActPos=> , 
	rActVelo=> , 
  );

  END_FOR	
 
  
IF  xRecipeAxisParSetButton THEN 
	FOR i:= 1 TO gc_uiAxisNum BY 1 DO
			stData.Axis[i].rAcceleration := 2000 ;
			stData.Axis[i].rDeceleration := 2000 ;
			stData.Axis[i].rJogVelocity := 10 ;
			stData.Axis[i].rManualVelocity := 20 ;
	    	stData.Axis[i].rAutoVelocity := 30;
	END_FOR
	xRecipeAxisParSetButton := FALSE ;
END_IF



//设定轴是直线定位还是模值定位
FOR i:= 1 TO 10 BY 1 DO 
	IF  i=9 OR i=14 THEN 
	fbAxis[i].xIsLinearMode := FALSE ;
	ELSE
	fbAxis[i].xIsLinearMode := TRUE ;
	END_IF
END_FOR
//设定模值模式时轴的路径(
(*fbAxis[5].nModuloDirection :=*)
fbAxis[9].nModuloDirection := 
fbAxis[14].nModuloDirection := MC_Direction.MC_Positive_Direction ;


//步进电机
fbAxis[17].xIRelative_Encoder:=TRUE;
fbAxis[18].xIRelative_Encoder:=TRUE;
fbAxis[19].xIRelative_Encoder:=TRUE;
END_ACTION

ACTION ACT_AxisHome:
sEctNetId := '192.168.1.1.2.1' ;//填写NETID
//回原点方式设定
home_method[1] :=27;
home_method[2] := 27 ;//35=机械回原点 23=正方向找原点 27=反方向找原点 7 11\
home_method[3] :=23;
home_method[4] := 27;
home_method[5] :=23;
home_method[6] := 27 ;
home_method[7] :=23;
home_method[8] := 27;
home_method[9] :=23;
home_method[10] := 23 ;
home_method[11] :=23;
home_method[12] := 23;
home_method[13] :=27;
home_method[14] := 27 ;
home_method[15] :=27;
home_method[16] := 23;



home_method[17] :=27;
fbAxisHome[17].iMode :=3;//雷赛伺服
home_method[18] :=27;
fbAxisHome[18].iMode :=3;
home_method[19] :=23;
fbAxisHome[19].iMode :=3;



//从站地址
cnSlaveAddr[01] := 1014 ;
cnSlaveAddr[02] := 1015 ;
cnSlaveAddr[03] := 1016 ;
cnSlaveAddr[04] := 1017 ;
cnSlaveAddr[05] := 1018 ;
cnSlaveAddr[06] := 1019 ;
cnSlaveAddr[07] := 1020 ;
cnSlaveAddr[08] := 1021 ;

cnSlaveAddr[09] := 1025 ;

cnSlaveAddr[10] := 1037 ;
cnSlaveAddr[11] := 1038 ;
cnSlaveAddr[12] := 1039 ;
cnSlaveAddr[13] := 1040 ;
cnSlaveAddr[14] := 1041 ;
cnSlaveAddr[15] := 1042 ;
cnSlaveAddr[16] := 1043 ;
cnSlaveAddr[17] := 1044 ;
cnSlaveAddr[18] := 1045 ;
cnSlaveAddr[19] := 1046 ;




FOR  i:=1 TO gc_uiAxisNum BY 1 DO
	IF i<=15 THEN
	fbAxisHome[i].home_highspeed_set:= 150; //
	fbAxisHome[i].home_lowspeed_set:= 5;
	fbAxisHome[i].numerator:=60;
	ELSIF i=16 THEN 
	 fbAxisHome[i].home_highspeed_set:= 40; //
	 fbAxisHome[i].home_lowspeed_set:= 5;
	 fbAxisHome[i].numerator:=60;
	else
		fbAxisHome[i].home_highspeed_set:=5; //雷赛
		fbAxisHome[i].home_lowspeed_set:= 1;
		fbAxisHome[i].numerator:=2;
	END_IF
		fbAxisHome[i].tTimeOutSet := T#60S;//超时时间设定
END_FOR


FOR  i:=1  TO gc_uiAxisNum BY 1 DO
 

		fbReference_TRIG[i](CLK:=fbAxis[i].xReferenceHmi OR  fbAxis[i].xReferenceAuto , Q=> );
		IF    fbReference_TRIG[i].Q THEN
			fbAxisHome[i].home_exe:=TRUE;
			fbAxis[i].xReferenceHmi :=FALSE;
		  fbAxis[i].xReferenceAuto:=FALSE;
		END_IF
		IF  fbAxisHome[i].home_exe AND   fbAxisHome[i].home_start THEN
		 			fbAxisHome[i].home_exe:=FALSE;
		END_IF
		fbAxisHome[i](
	    axis_name :=Axis[i], 
		home_exe:=,//fbAxis[i].xReferenceHmi OR  fbAxis[i].xReferenceAuto, 
		fb_netid:=sEctNetId , 
		fb_nslaveaddr:= cnSlaveAddr[i] , 
	    nctrl1:= nctrl1[i], 
	    nctrl2:= nctrl2[i], 		
	    mode:= sModeOperation[i],
        home_method := home_method[i],	
	    home_highspeed_set:= , 
	    home_lowspeed_set:= , 
	    home_offset_set:= 0,
	    numerator:= , 
	    denominator:= 4194304, 
		home_done=> , 
		home_error=> , 
 	    controlword=> controlword[i], 
	    error_id=> );

END_FOR








 
IF NOT bAxisHome_First THEN	
	FOR i:=1 TO  gc_uiAxisNum BY 1 DO	
	  sModeOperation[i] := 8;
	END_FOR
	bAxisHome_First := TRUE;
END_IF
//超时时间设定
END_ACTION

ACTION ACT_Camera:
FOR  i:= 1  TO gc_uiCameraNum   BY 1  DO 
	fbCamera[i](
		xlInit:= , 
		xlTrigger:= , 
		xlTriggerHmi:= , 
		xlLight:= TRUE, 
		xlReady:=TRUE , 
		xlAutoMode:=fbMachine[1].xAutoMode , 
		xlManualMode:=fbMachine[1].xManualMode  , 
		xITryRun:=fbMachine[1].xTryRun OR	axBypassSignal[3] , 
		tlDelay:= stData.Camera[i].tDelay, 
		xIDeviceRunning:=,
		xQStart=> , 
		xQLight=> , 
		xQCompleted=> , 
		xQAlarm=> , 
		xQBusy=> , 
		xQHmiAlarm=> , 
		ilCompleted:=sCamera_To_PLC.iCompleted[i]);
		
		//延时设定
		fbCamera[i].tlDelay:=fbCamera[1].tlDelay;
END_FOR


//上料工位相机光源触发
IF   fbCamera[1].xQLight  THEN
			QxCameraLight1Trigger:=TRUE;
			QxCameraLight2Trigger:=TRUE;
ELSE
 			QxCameraLight1Trigger:=FALSE;
			QxCameraLight2Trigger:=FALSE;
END_IF
//相机触发
QxCamera1Trigger:=fbCamera[1].xQStart;




//S03液位检测工位光源触发
IF 			fbCamera[2].xQLight OR	fbCamera[3].xQLight OR
				fbCamera[4].xQLight OR	fbCamera[5].xQLight OR
			  fbCamera[6].xQLight OR	fbCamera[7].xQLight OR
				fbCamera[8].xQLight OR	fbCamera[9].xQLight OR
			 fbCamera[10].xQLight OR	fbCamera[11].xQLight OR
			 fbCamera[12].xQLight OR	fbCamera[13].xQLight OR
			 fbCamera[14].xQLight OR	fbCamera[15].xQLight OR
				fbCamera[17].xQLight THEN
					QxCameraLight3Trigger:=TRUE;	
ELSE
 						QxCameraLight3Trigger:=FALSE;	
END_IF 
						 
//相机触发
QxCamera2Trigger	:= fbCamera[2].xQStart; 
QxCamera3Trigger	:= fbCamera[3].xQStart; 
QxCamera4Trigger	:= fbCamera[4].xQStart; 
QxCamera5Trigger	:= fbCamera[5].xQStart; 
QxCamera6Trigger	:= fbCamera[6].xQStart; 
QxCamera7Trigger	:= fbCamera[7].xQStart; 
QxCamera8Trigger	:= fbCamera[8].xQStart; 
QxCamera9Trigger	:= fbCamera[9].xQStart; 
QxCamera10Trigger   := fbCamera[10].xQStart; 
QxCamera11Trigger   := fbCamera[11].xQStart;
QxCamera12Trigger   := fbCamera[12].xQStart;
QxCamera13Trigger   := fbCamera[13].xQStart;
QxCamera14Trigger   := fbCamera[14].xQStart;
QxCamera15Trigger   := fbCamera[15].xQStart;
QxCamera16Trigger   := fbCamera[16].xQStart;
QxCamera17Trigger   := fbCamera[17].xQStart;
//贴标工位相机光源触发
IF  fbCamera[18].xQLight  THEN
 			QxCameraLight4Trigger:=TRUE;
ELSE
 			QxCameraLight4Trigger:=FALSE;
END_IF

//相机触发
QxCameraTrigger	:= fbCamera[18].xQStart; 


//相机型号
sCamera_From_Plc.iBoxType:=iBoxChoose;
END_ACTION

ACTION ACT_Cimcor:
FOR  i:= 1  TO gc_uiCimcorNum   BY 1  DO 
	fbCimcor[i](
	xIStart:= , 
	xIStop:= , 
	xIReset:= , 
	xICimcorMaint:= , 
	xIError:= , 
	xICimcorStarted:= , 
	xQError=> , 
	xQCimcorStart=> , 
	xQCimcorReset=> , 
	xQValveStart=> , 
	xQNeedMaint=> );
END_FOR
//离子风棒已开启
fbCimcor[1].xICimcorStarted:=IxStartSignal;
fbCimcor[1].xICimcorMaint:=IxMaintenanceSignal_1;//	卡片搬运工位¶离子风棒¶维护信号
fbCimcor[1].xIError:= NOT  IxErrorSignal_1;//	卡片搬运工位¶离子风棒¶异常信号

QxET02IonResetControl:=fbCimcor[1].xQCimcorReset;//	卡片搬运工位¶离子风棒¶复位信号
QxET02IonStopControl:=fbCimcor[1].xQCimcorStart;//卡片搬运工位¶离子风棒¶停止放电信号
										
//QxET02IonControlSignal1	:BOOL;//	卡片搬运工位¶离子风棒¶外部给定信号1
//QxET02IonControlSignal2	:BOOL;//	卡片搬运工位¶离子风棒¶外部给定信号2
//电磁阀控制
QxS09ControlValve:=fbCimcor[1].xQValveStart;//	卡片工位离子风棒气路控制
END_ACTION

ACTION ACT_Comm:
//(*************************** Clock 1 Second Clock***********************************)
//tTonoff1s(IN:=NOT tTonOn1s.Q,PT:=T#1S);
//
//tTonOn1s(IN:= tTonOff1s.Q,PT:=T#1S);
//
//(****************************Alive bit************************************)
//IF  tTonoff1s.Q THEN
//	 sPLC_TO_PC.xPLCALive:=1 ;
//	
//ELSE
//	 sPLC_TO_PC.xPLCALive:=0;
//END_IF
END_ACTION

ACTION ACT_Cylinder:
//上电复位
IF NOT xCylinder_First THEN
  FOR i :=1 TO gc_uiCylinderNum DO 
    fbCylinder[i].xHmi               :=FALSE;	 
  END_FOR
 	 xCylinder_First                :=TRUE;
END_IF


FOR i:= 1 TO gc_uiCylinderNum BY 1 DO 
fbCylinder[i](
	xEStop:=fbMachine[1].xEStop,  
	xSafety:=fbMachine[1].xSafety , 
	xManualMode:=fbMachine[1].xManualMode , 
	xAutoMode:=fbMachine[1].xAutoMode , 
	xAirOn:=fbMachine[1].xAirOn , 
	tAlarm:=stData.Cylinder[i].Alarm_Delay , 
	xReset:=fbMachine[1].xReset , 
	xTryRun:= fbmachine[1].xTryRun, 
	xAlarmDisable:= , 
	xHmi:= , 
	tHP_Delay:=stData.Cylinder[i].tHP_Delay , 
	tWP_Delay:=stData.Cylinder[i].tWP_Delay ,  
	xHP_Valve=> , 
	xWP_Valve=> , 
	xHP_Delay=> , 
	xWP_Delay=> );
END_FOR
END_ACTION

ACTION ACT_EasyPump:
fbEasyPumps[1].LocalClient.strSlaveIP:='192.168.1.60';
fbEasyPumps[1].LocalClient.iSlavePort:=1031;
fbEasyPumps[1].LocalClient.bySlaveID:=1;

fbEasyPumps[2].LocalClient.strSlaveIP:='192.168.1.61';
fbEasyPumps[2].LocalClient.iSlavePort:=1031;
fbEasyPumps[2].LocalClient.bySlaveID:=1;

fbEasyPumps[3].LocalClient.strSlaveIP:='192.168.1.62';
fbEasyPumps[3].LocalClient.iSlavePort:=1031;
fbEasyPumps[3].LocalClient.bySlaveID:=1;

fbEasyPumps[4].LocalClient.strSlaveIP:='192.168.1.63';
fbEasyPumps[4].LocalClient.iSlavePort:=1031;
fbEasyPumps[4].LocalClient.bySlaveID:=1;

fbEasyPumps[5].LocalClient.strSlaveIP:='192.168.1.66';
fbEasyPumps[5].LocalClient.iSlavePort:=1031;
fbEasyPumps[5].LocalClient.bySlaveID:=1;

fbEasyPumps[6].LocalClient.strSlaveIP:='192.168.1.65';
fbEasyPumps[6].LocalClient.iSlavePort:=1031;
fbEasyPumps[6].LocalClient.bySlaveID:=1;

fbEasyPumps[7].LocalClient.strSlaveIP:='192.168.1.67';
fbEasyPumps[7].LocalClient.iSlavePort:=1031;
fbEasyPumps[7].LocalClient.bySlaveID:=1;

fbEasyPumps[8].LocalClient.strSlaveIP:='192.168.1.68';
fbEasyPumps[8].LocalClient.iSlavePort:=1031;
fbEasyPumps[8].LocalClient.bySlaveID:=1;

fbEasyPumps[9].LocalClient.strSlaveIP:='192.168.1.69';
fbEasyPumps[9].LocalClient.iSlavePort:=1031;
fbEasyPumps[9].LocalClient.bySlaveID:=1;

fbEasyPumps[10].LocalClient.strSlaveIP:='192.168.1.71';
fbEasyPumps[10].LocalClient.iSlavePort:=1031;
fbEasyPumps[10].LocalClient.bySlaveID:=1;

fbEasyPumps[11].LocalClient.strSlaveIP:='192.168.1.70';
fbEasyPumps[11].LocalClient.iSlavePort:=1031;
fbEasyPumps[11].LocalClient.bySlaveID:=1;

fbEasyPumps[12].LocalClient.strSlaveIP:='192.168.1.64';
fbEasyPumps[12].LocalClient.iSlavePort:=1031;
fbEasyPumps[12].LocalClient.bySlaveID:=1;


//如果泵参数固定，就直接配置好，如果不固定，就在触摸屏配置
stData.EasyPumps[1].iPumpType:=stEasyPumpType.i_DFPluse;//设定泵控制器类型
stData.EasyPumps[1].iPumpTypeSet:=stEasyPumpHeadType.i_MiniPump01;//设定泵泵头类型
stData.EasyPumps[1].iHosePipeTypeSet:=RudongPump_SoftPipeType.P19;//设定泵软管类型
//如果泵参数固定，就直接配置好，如果不固定，就在触摸屏配置
stData.EasyPumps[2].iPumpType:=stEasyPumpType.i_DFPluse;//设定泵控制器类型
stData.EasyPumps[2].iPumpTypeSet:=stEasyPumpHeadType.i_MiniPump01;//设定泵泵头类型
stData.EasyPumps[2].iHosePipeTypeSet:=RudongPump_SoftPipeType.P19;//设定泵软管类
//如果泵参数固定，就直接配置好，如果不固定，就在触摸屏配置
stData.EasyPumps[3].iPumpType:=stEasyPumpType.i_DFPluse;//设定泵控制器类型
stData.EasyPumps[3].iPumpTypeSet:=stEasyPumpHeadType.i_MiniPump01;//设定泵泵头类型
stData.EasyPumps[3].iHosePipeTypeSet:=RudongPump_SoftPipeType.P19;//设定泵软管类型
//如果泵参数固定，就直接配置好，如果不固定，就在触摸屏配置
stData.EasyPumps[4].iPumpType:=stEasyPumpType.i_DFPluse;//设定泵控制器类型
stData.EasyPumps[4].iPumpTypeSet:=stEasyPumpHeadType.i_MiniPump01;//设定泵泵头类型
stData.EasyPumps[4].iHosePipeTypeSet:=RudongPump_SoftPipeType.P19;//设定泵软管类型
//如果泵参数固定，就直接配置好，如果不固定，就在触摸屏配置
stData.EasyPumps[5].iPumpType:=stEasyPumpType.i_DFPluse;//设定泵控制器类型
stData.EasyPumps[5].iPumpTypeSet:=stEasyPumpHeadType.i_MiniPump01;//设定泵泵头类型
stData.EasyPumps[5].iHosePipeTypeSet:=RudongPump_SoftPipeType.P19;//设定泵软管类型
//如果泵参数固定，就直接配置好，如果不固定，就在触摸屏配置
stData.EasyPumps[6].iPumpType:=stEasyPumpType.i_DFPluse;//设定泵控制器类型
stData.EasyPumps[6].iPumpTypeSet:=stEasyPumpHeadType.i_HandyPump01;//设定泵泵头类型
stData.EasyPumps[6].iHosePipeTypeSet:=RudongPump_SoftPipeType.P13;//设定泵软管类型
//如果泵参数固定，就直接配置好，如果不固定，就在触摸屏配置
stData.EasyPumps[7].iPumpType:=stEasyPumpType.i_DFPluse;//设定泵控制器类型
stData.EasyPumps[7].iPumpTypeSet:=stEasyPumpHeadType.i_MiniPump01;//设定泵泵头类型
stData.EasyPumps[7].iHosePipeTypeSet:=RudongPump_SoftPipeType.P19;//设定泵软管类型
//如果泵参数固定，就直接配置好，如果不固定，就在触摸屏配置
stData.EasyPumps[8].iPumpType:=stEasyPumpType.i_DFPluse;//设定泵控制器类型
stData.EasyPumps[8].iPumpTypeSet:=stEasyPumpHeadType.i_MiniPump01;//设定泵泵头类型
stData.EasyPumps[8].iHosePipeTypeSet:=RudongPump_SoftPipeType.P19;//设定泵软管类型
//如果泵参数固定，就直接配置好，如果不固定，就在触摸屏配置
stData.EasyPumps[9].iPumpType:=stEasyPumpType.i_DFPluse;//设定泵控制器类型
stData.EasyPumps[9].iPumpTypeSet:=stEasyPumpHeadType.i_MiniPump01;//设定泵泵头类型
stData.EasyPumps[9].iHosePipeTypeSet:=RudongPump_SoftPipeType.P19;//设定泵软管类型
//如果泵参数固定，就直接配置好，如果不固定，就在触摸屏配置
stData.EasyPumps[10].iPumpType:=stEasyPumpType.i_DFPluse;//设定泵控制器类型
stData.EasyPumps[10].iPumpTypeSet:=stEasyPumpHeadType.i_MiniPump01;//设定泵泵头类型
stData.EasyPumps[10].iHosePipeTypeSet:=RudongPump_SoftPipeType.P19;//设定泵软管类型
//如果泵参数固定，就直接配置好，如果不固定，就在触摸屏配置
stData.EasyPumps[11].iPumpType:=stEasyPumpType.i_DFPluse;//设定泵控制器类型
stData.EasyPumps[11].iPumpTypeSet:=stEasyPumpHeadType.i_MiniPump01;//设定泵泵头类型
stData.EasyPumps[11].iHosePipeTypeSet:=RudongPump_SoftPipeType.P19;//设定泵软管类型
//如果泵参数固定，就直接配置好，如果不固定，就在触摸屏配置
stData.EasyPumps[12].iPumpType:=stEasyPumpType.i_DFPluse;//设定泵控制器类型
stData.EasyPumps[12].iPumpTypeSet:=stEasyPumpHeadType.i_HandyPump01;//设定泵泵头类型
stData.EasyPumps[12].iHosePipeTypeSet:=RudongPump_SoftPipeType.P13;//设定泵软管类型

///方向设定
stData.EasyPumps[1].iDirectionSet:=1;
stData.EasyPumps[2].iDirectionSet:=0;
stData.EasyPumps[3].iDirectionSet:=1;
stData.EasyPumps[4].iDirectionSet:=0;
stData.EasyPumps[5].iDirectionSet:=1;
stData.EasyPumps[6].iDirectionSet:=0;
stData.EasyPumps[7].iDirectionSet:=0;
stData.EasyPumps[8].iDirectionSet:=1;
stData.EasyPumps[9].iDirectionSet:=0;
stData.EasyPumps[10].iDirectionSet:=1;
stData.EasyPumps[11].iDirectionSet:=0;
stData.EasyPumps[12].iDirectionSet:=1;



stData.EasyPumps[1].iAccuracySet:=0.03;
stData.EasyPumps[2].iAccuracySet:=0.03;
stData.EasyPumps[3].iAccuracySet:=0.03;
stData.EasyPumps[4].iAccuracySet:=0.03;
stData.EasyPumps[5].iAccuracySet:=0.03;
stData.EasyPumps[6].iAccuracySet:=0.065;
stData.EasyPumps[7].iAccuracySet:=0.03;
stData.EasyPumps[8].iAccuracySet:=0.03;
stData.EasyPumps[9].iAccuracySet:=0.03;
stData.EasyPumps[10].iAccuracySet:=0.03;
stData.EasyPumps[11].iAccuracySet:=0.03;
stData.EasyPumps[12].iAccuracySet:=0.065;

FOR i:=1 TO gc_uiRudongPump BY 1 DO
 		IF  fbMachine[1].xReset THEN
 			  fbEasyPumps[i].xIReset:=TRUE;
	  END_IF
 		fbEasyPumps[i](
							xIReset:= , 
							xIManualMode:=fbMachine[1].xManualMode, 
							xIAutoMode:= fbMachine[1].xAutoMode, 
							xIEstop:= NOT fbMachine[1].xEStop,
							xIDeviceRunning:=TRUE, 
							stRunPara:= stData.EasyPumps[i], 
							stDeviceOpe:= , 
							xQBusy=> , 
							xQDone=> , 
							rMaxRunTime=> , 
							rMinRunTime=> );
END_FOR
END_ACTION

ACTION ACT_Encoder:
fbEncoder(
	xIErrorReset:= , 
	tDelay:=T#500MS, 
	xQBusy=> , 
	xQError=> , 
	iQErrorNo=> , 
	rQBeltSpeed=> );
END_ACTION

ACTION ACT_ERG_20C:
	fbERG[1].LocalClient.bySlaveID := 1;
	fbERG[1].LocalClient.strSlaveIP := '192.168.1.20';//从站IP地址
	fbERG[1].LocalClient.iSlavePort := 1030;	//四端口智嵌物联
	
	fbERG[2].LocalClient.bySlaveID := 1;
	fbERG[2].LocalClient.strSlaveIP := '192.168.1.21';//从站IP地址
	fbERG[2].LocalClient.iSlavePort := 1031;


FOR i:=1 TO gc_uiHITBOT_Number BY 1 DO
	IF fbMachine[1].xReset THEN
			  fbERG[i].xIReset:=TRUE;
	END_IF
 fbERG[i](
	xIReset:= , 
	xIManualMode:= fbMachine[1].xManualMode, 
	xIAutoMode:= fbMachine[1].xAutoMode, 
	xIDeviceRunning:=TRUE ,
	stRunPara:=stData.ERG20C[i] , 
	stDeviceOpe:= , 
	stDevice=> , 
	stPara=> , 
	stReadPara=> , 
	iQErrorID=> , 
	strQErrorID=> );
END_FOR

stData.ERG20C[1].aHMIClampPara[1].rCurrentSet:=0.4;
stData.ERG20C[1].aHMIClampPara[1].rPositionSet:=5;
stData.ERG20C[1].aHMIClampPara[1].rSpeedSet:=200;
stData.ERG20C[1].aHMIReleasePara[1].rCurrentSet:=0.4;
stData.ERG20C[1].aHMIReleasePara[1].rPositionSet:=15;
stData.ERG20C[1].aHMIReleasePara[1].rSpeedSet:=200;


stData.ERG20C[1].aHMIRotateClampPara[1].rCurrentSet:=0.5;
stData.ERG20C[1].aHMIRotateClampPara[1].rPositionSet:=180;
stData.ERG20C[1].aHMIRotateClampPara[1].rSpeedSet:=500;

stData.ERG20C[1].aHMIRotateReleasePara[1].rCurrentSet:=0.5;
stData.ERG20C[1].aHMIRotateReleasePara[1].rPositionSet:=0;
stData.ERG20C[1].aHMIRotateReleasePara[1].rSpeedSet:=300;

stData.ERG20C[2].aHMIClampPara[1].rCurrentSet:=0.4;
stData.ERG20C[2].aHMIClampPara[1].rPositionSet:=5;
stData.ERG20C[2].aHMIClampPara[1].rSpeedSet:=200;
stData.ERG20C[2].aHMIReleasePara[1].rCurrentSet:=0.4;
stData.ERG20C[2].aHMIReleasePara[1].rPositionSet:=15;
stData.ERG20C[2].aHMIReleasePara[1].rSpeedSet:=200;


stData.ERG20C[2].aHMIRotateClampPara[1].rCurrentSet:=0.9;
stData.ERG20C[2].aHMIRotateClampPara[1].rPositionSet:=180;
stData.ERG20C[2].aHMIRotateClampPara[1].rSpeedSet:=500;

stData.ERG20C[2].aHMIRotateReleasePara[1].rCurrentSet:=0.6;
stData.ERG20C[2].aHMIRotateReleasePara[1].rPositionSet:=0;
stData.ERG20C[2].aHMIRotateReleasePara[1].rSpeedSet:=300;
END_ACTION

ACTION ACT_EtherCATSlaveState:

(****************************************************Error Pause****************************************************)
(* EtherCAT Terminal error*)
FOR   i:=1 TO gc_uiSlaveNum BY 1 DO
fbEhterCATSlaveMonitor[i](
	xIActive:=TRUE ,
	xIReset:=fbMachine[1].xReset,
	axIState:= ,
	xQError=> ,
	iQErrorTerm=> );
END_FOR
END_ACTION

ACTION ACT_FuShiPXF:
IF ( NOT _firstFuShiPXF) THEN
fbTempretureControl[1].stSysPar.strSlaveIP:='192.168.1.90';
fbTempretureControl[1].stSysPar.bySlaveID:=2;
fbTempretureControl[1].stSysPar.iSlavePort:=1032;
fbTempretureControl[2].stSysPar.strSlaveIP:='192.168.1.90';
fbTempretureControl[2].stSysPar.bySlaveID:=3;
fbTempretureControl[2].stSysPar.iSlavePort:=1033;
 _firstFuShiPXF := TRUE;
ELSE
FOR i:=1 TO gc_uiPXF5Num DO
fbTempretureControl[i](
	xEstop:= fbMachine[1].xEStop , 
	xStart:= , 
	xSvSet:= , 
	stSysPar:= , 
	stPar:= , 
	stParRead=> , 
	xRdy=> , 
	xPowerOut=> , 
	xError=> , 
	sError=> );
END_FOR

END_IF
//温控器控制加热棒使能
QxHeatRelayContorl1:=fbTempretureControl[1].xPowerOut;
QxHeatRelayContorl2:=fbTempretureControl[2].xPowerOut;

//QxEnableHeatingRod:=fbTempretureControl[1].xPowerOut AND fbTempretureControl[2].xPowerOut;
//S04_FilmCovering.xHeatingDeviceReady:=fbTempretureControl[1].xRdy AND fbTempretureControl[2].xRdy;
END_ACTION

ACTION ACT_GetTime:
PRG_GetSystemTime();

strLocalDateTime := SYSTEMTIME_TO_STRING(PRG_GetSystemTime.sQTime);
strDateTime := MID( strLocalDateTime,8,12 ) ;

stDateTime.sTempTimeYYMMDD:= MID (strLocalDateTime, 11, 1 );
stDateTime.sTempTimeHO:= MID (strLocalDateTime, 2, 12 );
stDateTime.sTempTimeMI:= MID (strLocalDateTime, 2, 15 );
stDateTime.sTempTimeSe:= MID (strLocalDateTime, 2, 18 );


FBGetTime(
	i_b_start:= , 
	i_b_withoutHs:= , 
	o_b_ok=> , 
	o_b_err=> , 
	o_udi_ErrId=> , 
	o_DateAndTime=> );
END_ACTION

ACTION ACT_LoadCell:
fbLoadCell[1].LocalClient.strSlaveIP:='192.168.1.73';
fbLoadCell[1].LocalClient.iSlavePort:=1030;
fbLoadCell[1].LocalClient.bySlaveID:=1;

fbLoadCell[2].LocalClient.strSlaveIP:='192.168.1.73';
fbLoadCell[2].LocalClient.iSlavePort:=1031;
fbLoadCell[2].LocalClient.bySlaveID:=2;

fbLoadCell[3].LocalClient.strSlaveIP:='192.168.1.74';
fbLoadCell[3].LocalClient.iSlavePort:=1030;
fbLoadCell[3].LocalClient.bySlaveID:=3;

fbLoadCell[4].LocalClient.strSlaveIP:='192.168.1.74';
fbLoadCell[4].LocalClient.iSlavePort:=1031;
fbLoadCell[4].LocalClient.bySlaveID:=4;


fbLoadCell[5].LocalClient.strSlaveIP:='192.168.1.75';
fbLoadCell[5].LocalClient.iSlavePort:=1030;
fbLoadCell[5].LocalClient.bySlaveID:=5;


fbLoadCell[6].LocalClient.strSlaveIP:='192.168.1.75';
fbLoadCell[6].LocalClient.iSlavePort:=1031;
fbLoadCell[6].LocalClient.bySlaveID:=6;



FOR i:=1 TO gc_uiLoadcellNum  DO
	fbLoadCell[i](
	xIStart:= , 
	xIReset:= , 
	LocalClient:= , 
	stDeviceOpe:= , 
	xIDeviceRunning:=TRUE , 
	xManualMode:= fbMachine[1].xManualMode, 
	xAutoMode:= fbMachine[1].xAutoMode, 
	xQRdyCmd=> , 
	xQBusy=> , 
	xQError=> , 
	xQDone=> , 
	stParOut=> );
END_FOR
//清零或去皮信号
QxLoadCell_1ZeroInput:=fbLoadCell[1].xQZeroSingle;
QxLoadCell_2ZeroInput:=fbLoadCell[2].xQZeroSingle;
QxLoadCell_3ZeroInput:=fbLoadCell[3].xQZeroSingle;
QxLoadCell_4ZeroInput:=fbLoadCell[4].xQZeroSingle;
QxLoadCell_5ZeroInput:=fbLoadCell[5].xQZeroSingle;
QxLoadCell_6ZeroInput:=fbLoadCell[6].xQZeroSingle;
END_ACTION

ACTION ACT_M0dbus_200Smart:
fbModbus_200Smart.stPara.strSlaveIP:='192.168.1.2';
fbModbus_200Smart.stPara.iSlavePort:=502;
fbModbus_200Smart.stPara.bySlaveID:=1;
fbModbus_200Smart(stPara:= , pSysTo200Smart:= , pSysFrom200Smart:= , st_IOData:=sModbus_200SMART );
//Output-Mapping
IF  fbMachine[1].xManualMode THEN
sModbus_200SMART.iMachineMode:=1;
ELSIF fbMachine[1].xAutoMode THEN
sModbus_200SMART.iMachineMode:=2;
END_IF
IF  fbMachine[1].xRunning THEN 
sModbus_200SMART.iMachineStart:=1;
END_IF 
IF fbMachine[1].xStop OR fbMachine[1].xPause THEN 
sModbus_200SMART.iMachineStop:=1;
ELSE
 sModbus_200SMART.iMachineStop:=0;
END_IF
IF  fbMachine[1].xIniting THEN 
	sModbus_200SMART.iMachineIniting:=1 ;
ELSE
	sModbus_200SMART.iMachineIniting:=0 ;
END_IF
IF fbStation[11].xDisabled THEN  
	sModbus_200SMART.iMachineDisable:=1 ;
ELSE
 sModbus_200SMART.iMachineDisable:=1 ;
END_IF
END_ACTION

ACTION ACT_Machine:


FOR i:=1 TO gc_uiMachineNum DO
fbMachine[i](
	xEmptyHmi:= , 
	xTryRun:= , 
	xEmptyConfirmHmi:= , 
	xInitConfirm:= ,
  xStart:= IxStartButton OR fbProface[1].xStartHmi ,
  xStop:= IxStopButton OR fbProface[1].xStopHmi ,
  xReset:= IxResetButton OR fbProface[1].xResetHmi ,
  xPause:= IxStopButton OR fbProface[1].xPauseHmi ,
  xInit:=IxInitButton OR fbProface[1].xInitHmi ,
  xManualMode:= (IxManualMode ), 
  xAutoMode:= ( IxAutoMode ) ,	 
	xRunning=>  , 
	xEmptying=> ,
	xEStopped=> , 
	xIniting=>  , 
	diCycleTime => ,
	xStopped=> , 
	xPaused=> , 	
   );
	END_FOR
QxRedLamp:=
QxRedLamp_1	 :=fbMachine[1].xLampRed;	
QxYellowLamp:=
QxYellowLamp_1 :=fbMachine[1].xLampYellow 	;///初始化完成后也需要将黄灯常亮
QxGreenLamp:=
QxGreenLamp_1 :=fbMachine[1].xLampGreen;	
IF  NOT   _BuzzerBypassButton  THEN
	QxBuzzer:=fbMachine[1].xLampBuzzer;
ELSE
	QxBuzzer:=FALSE;
END_IF
IF  _BuzzerBypassButton THEN
	_BuzzerBypassLamp:=TRUE;
ELSE
	_BuzzerBypassLamp:=FALSE;
END_IF
QxStartButtonLamp	:=fbMachine[1].xStartLight;
QxStopButtonLamp	:=fbMachine[1].xStopLight;	
QxResetButtonLamp	:=fbMachine[1].xResetLight;	
QxInitButtonLamp	:=fbMachine[1].xInitLight;
END_ACTION

ACTION ACT_MT_MCK:
fbMCK204W.stSysPar.sRemoteHost:='192.168.1.72';
fbMCK204W.stSysPar.nRemotePort:=1030;
fbMCK204W.stSysPar.bySlaveID:=1;
fbMCK204W.xDeviceRunning:=fbAutoCal.xRunning;
fbMCK204W(
	xExecute:= , 
	xAbort:= , 
	xEstop:=  fbMachine[1].xEStop, 
	xDeviceRunning:= , 
	xResetRequest:= , 
	stDeviceOpe:= , 
	stpar:= , 
	stSysPar:= , 
	dwTimeOut:= , 
	xManualHMIControl:= , 
	xAutoMode:= , 
	xIniting:= , 
	xDone=> , 
	xBusy=> , 
	xError=> , 
	eErrorID=> , 
	eTCPErrorID=> , 
	xRdyCmd=> , 
	xRefOk=> , 
	stParOut=> );
END_ACTION

ACTION ACT_MT_MCK_1:
fbMCK.stSysPar.sRemoteHost:='192.168.1.72';
fbMCK.stSysPar.nRemotePort:=1030;
fbMCK.stSysPar.bySlaveID:=1;

fbMCK(
	xIReset:=(*fbMachine[1].xReset*) , 
	xIInit:= , 
	iICodeLEN:= 20, 
	iICodePOS:= 1, 
	xIDeviceRunning:= TRUE, 
	xManualMode:=fbMachine[1].xManualMode , 
	xAutoMode:=fbMachine[1].xAutoMode , 
	stDeviceOpe:= , 
	stpar:= , 
	stSysPar:= , 
	xQRdyCmd=> , 
	xQDone=> , 
	strQBarCode=> , 
	xQBusy=> , 
	xQError=> , 
	xQNoRead=> , 
	iQErrorNo=> , 
	stParOut=> );
END_ACTION

ACTION ACT_PeristalticPump:
fbRudongPump[1].stPara.strSlaveIP:='192.168.1.60';
fbRudongPump[1].stPara.iSlavePort:=1031;
fbRudongPump[1].stPara.bySlaveID:=1;

fbRudongPump[2].stPara.strSlaveIP:='192.168.1.61';
fbRudongPump[2].stPara.iSlavePort:=1031;
fbRudongPump[2].stPara.bySlaveID:=1;

fbRudongPump[3].stPara.strSlaveIP:='192.168.1.62';
fbRudongPump[3].stPara.iSlavePort:=1031;
fbRudongPump[3].stPara.bySlaveID:=1;

fbRudongPump[4].stPara.strSlaveIP:='192.168.1.63';
fbRudongPump[4].stPara.iSlavePort:=1031;
fbRudongPump[4].stPara.bySlaveID:=1;

fbRudongPump[5].stPara.strSlaveIP:='192.168.1.66';
fbRudongPump[5].stPara.iSlavePort:=1031;
fbRudongPump[5].stPara.bySlaveID:=1;

fbRudongPump[6].stPara.strSlaveIP:='192.168.1.65';
fbRudongPump[6].stPara.iSlavePort:=1031;
fbRudongPump[6].stPara.bySlaveID:=1;

fbRudongPump[7].stPara.strSlaveIP:='192.168.1.67';
fbRudongPump[7].stPara.iSlavePort:=1031;
fbRudongPump[7].stPara.bySlaveID:=1;

fbRudongPump[8].stPara.strSlaveIP:='192.168.1.68';
fbRudongPump[8].stPara.iSlavePort:=1031;
fbRudongPump[8].stPara.bySlaveID:=1;

fbRudongPump[9].stPara.strSlaveIP:='192.168.1.69';
fbRudongPump[9].stPara.iSlavePort:=1031;
fbRudongPump[9].stPara.bySlaveID:=1;

fbRudongPump[10].stPara.strSlaveIP:='192.168.1.71';
fbRudongPump[10].stPara.iSlavePort:=1031;
fbRudongPump[10].stPara.bySlaveID:=1;

fbRudongPump[11].stPara.strSlaveIP:='192.168.1.70';
fbRudongPump[11].stPara.iSlavePort:=1031;
fbRudongPump[11].stPara.bySlaveID:=1;

fbRudongPump[12].stPara.strSlaveIP:='192.168.1.64';
fbRudongPump[12].stPara.iSlavePort:=1031;
fbRudongPump[12].stPara.bySlaveID:=1;

//如果泵参数固定，就直接配置好，如果不固定，就在触摸屏配置
stData.RudongPump[1].iPumpType:=RudongPump_PumpType.DFPluse;//设定泵控制器类型
stData.RudongPump[1].iPumpTypeSet:=RudongPump_PumpHeadType.MiniPump01;//设定泵泵头类型
stData.RudongPump[1].iHosePipeTypeSet:=RudongPump_SoftPipeType.P19;//设定泵软管类型
//如果泵参数固定，就直接配置好，如果不固定，就在触摸屏配置
stData.RudongPump[2].iPumpType:=RudongPump_PumpType.DFPluse;//设定泵控制器类型
stData.RudongPump[2].iPumpTypeSet:=RudongPump_PumpHeadType.MiniPump01;//设定泵泵头类型
stData.RudongPump[2].iHosePipeTypeSet:=RudongPump_SoftPipeType.P19;//设定泵软管类
//如果泵参数固定，就直接配置好，如果不固定，就在触摸屏配置
stData.RudongPump[3].iPumpType:=RudongPump_PumpType.DFPluse;//设定泵控制器类型
stData.RudongPump[3].iPumpTypeSet:=RudongPump_PumpHeadType.MiniPump01;//设定泵泵头类型
stData.RudongPump[3].iHosePipeTypeSet:=RudongPump_SoftPipeType.P19;//设定泵软管类型
//如果泵参数固定，就直接配置好，如果不固定，就在触摸屏配置
stData.RudongPump[4].iPumpType:=RudongPump_PumpType.DFPluse;//设定泵控制器类型
stData.RudongPump[4].iPumpTypeSet:=RudongPump_PumpHeadType.MiniPump01;//设定泵泵头类型
stData.RudongPump[4].iHosePipeTypeSet:=RudongPump_SoftPipeType.P19;//设定泵软管类型
//如果泵参数固定，就直接配置好，如果不固定，就在触摸屏配置
stData.RudongPump[5].iPumpType:=RudongPump_PumpType.DFPluse;//设定泵控制器类型
stData.RudongPump[5].iPumpTypeSet:=RudongPump_PumpHeadType.MiniPump01;//设定泵泵头类型
stData.RudongPump[5].iHosePipeTypeSet:=RudongPump_SoftPipeType.P19;//设定泵软管类型
//如果泵参数固定，就直接配置好，如果不固定，就在触摸屏配置
stData.RudongPump[6].iPumpType:=RudongPump_PumpType.DFPluse;//设定泵控制器类型
stData.RudongPump[6].iPumpTypeSet:=RudongPump_PumpHeadType.HandyPump01;//设定泵泵头类型
stData.RudongPump[6].iHosePipeTypeSet:=RudongPump_SoftPipeType.P13;//设定泵软管类型
//如果泵参数固定，就直接配置好，如果不固定，就在触摸屏配置
stData.RudongPump[7].iPumpType:=RudongPump_PumpType.DFPluse;//设定泵控制器类型
stData.RudongPump[7].iPumpTypeSet:=RudongPump_PumpHeadType.MiniPump01;//设定泵泵头类型
stData.RudongPump[7].iHosePipeTypeSet:=RudongPump_SoftPipeType.P19;//设定泵软管类型
//如果泵参数固定，就直接配置好，如果不固定，就在触摸屏配置
stData.RudongPump[8].iPumpType:=RudongPump_PumpType.DFPluse;//设定泵控制器类型
stData.RudongPump[8].iPumpTypeSet:=RudongPump_PumpHeadType.MiniPump01;//设定泵泵头类型
stData.RudongPump[8].iHosePipeTypeSet:=RudongPump_SoftPipeType.P19;//设定泵软管类型
//如果泵参数固定，就直接配置好，如果不固定，就在触摸屏配置
stData.RudongPump[9].iPumpType:=RudongPump_PumpType.DFPluse;//设定泵控制器类型
stData.RudongPump[9].iPumpTypeSet:=RudongPump_PumpHeadType.MiniPump01;//设定泵泵头类型
stData.RudongPump[9].iHosePipeTypeSet:=RudongPump_SoftPipeType.P19;//设定泵软管类型
//如果泵参数固定，就直接配置好，如果不固定，就在触摸屏配置
stData.RudongPump[10].iPumpType:=RudongPump_PumpType.DFPluse;//设定泵控制器类型
stData.RudongPump[10].iPumpTypeSet:=RudongPump_PumpHeadType.MiniPump01;//设定泵泵头类型
stData.RudongPump[10].iHosePipeTypeSet:=RudongPump_SoftPipeType.P19;//设定泵软管类型
//如果泵参数固定，就直接配置好，如果不固定，就在触摸屏配置
stData.RudongPump[11].iPumpType:=RudongPump_PumpType.DFPluse;//设定泵控制器类型
stData.RudongPump[11].iPumpTypeSet:=RudongPump_PumpHeadType.MiniPump01;//设定泵泵头类型
stData.RudongPump[11].iHosePipeTypeSet:=RudongPump_SoftPipeType.P19;//设定泵软管类型
//如果泵参数固定，就直接配置好，如果不固定，就在触摸屏配置
stData.RudongPump[12].iPumpType:=RudongPump_PumpType.DFPluse;//设定泵控制器类型
stData.RudongPump[12].iPumpTypeSet:=RudongPump_PumpHeadType.HandyPump01;//设定泵泵头类型
stData.RudongPump[12].iHosePipeTypeSet:=RudongPump_SoftPipeType.P13;//设定泵软管类型

///方向设定
fbRudongPump[1].iDirectionSet:=1;
fbRudongPump[2].iDirectionSet:=0;
fbRudongPump[3].iDirectionSet:=1;
fbRudongPump[4].iDirectionSet:=0;
fbRudongPump[5].iDirectionSet:=1;
fbRudongPump[6].iDirectionSet:=0;
fbRudongPump[7].iDirectionSet:=0;
fbRudongPump[8].iDirectionSet:=1;
fbRudongPump[9].iDirectionSet:=0;
fbRudongPump[10].iDirectionSet:=1;
fbRudongPump[11].iDirectionSet:=0;
fbRudongPump[12].iDirectionSet:=1;



FOR i :=1 TO gc_uiRudongPump BY 1 DO
	fbRudongPump[i](
	xExecute:= , 
	xAbort:= , 
	xResetRequest:=, 
	xRunILC:=TRUE , 
	dwTimeLimit:= , 
	dwTimeOut:= , 
	stPara:=, 
	xNeedConfigurePara:= , 
	stRunPara:=stData.RudongPump[i] , 
	xAutoMode:=fbMachine[1].xAutoMode , 
	xIniting:= , 
	xDeviceRunning:= , 
	rSpeedRatio:= , 
	sHmiError:= , 
	xEStop:= fbMachine[1].xEStop , 
	stDeviceOpe:= , 
	xDone=> , 
	xBusy=> , 
	xError=> , 
	xAborted=> , 
	xRunning=> , 
	xRudongPump_ERROR=> , 
	eERRORID=> , 
	xRdyCmd=> );
	
	//确定蠕动泵注液方向
	IF  fbMachine[1].xManualMode THEN
			 IF i MOD 2  = 0 THEN 
							 fbRudongPump[i].iDirectionSet:=0;
			 ELSE
							 fbRudongPump[i].iDirectionSet:=1;
			 END_IF
	END_IF
END_FOR
//IF NOT _xCalFirstCycle THEN
////	fbAutoCal.stSysPar.fbMTMCK204C:=ADR	(fbMCK204W);
//	fbAutoCal.stSysPar.fbMTMCK204C:=ADR	(fbMCK);
//	fbAutoCal.stSysPar.fbRuDongPump:=ADR(fbRudongPump[1]);
//	fbAutoCal.stparIn.iContinuesInjectNum:=5;//连续加液次数
//	fbAutoCal.stparIn.rDensity:=1;//密度为1
//	fbAutoCal.stparIn.tSteadyTime:=5;//稳定5秒
//	fbAutoCal.stparIn.iPumpController:=1;//控制器个数
//	_xCalFirstCycle:=TRUE;
//ELSE
//	fbAutoCal(
//		xExecute:= , 
//		xAbort:= , 
//		xEstop:= fbMachine[1].xEStop, 
//		xDeviceRunning:= , 
//		xResetRequest:= , 
//		stDeviceOpe:= , 
//		stparIn:= , 
//		stSysPar:= , 
//		xAutoMode:= , 
//		xIniting:= , 
//		xDone=> , 
//		xBusy=> , 
//		xError=> , 
//		eERRORID=> , 
//		xRdyCmd=> , 
//		xRdy=> , 
//		stParOut=> );	
//END_IF
END_ACTION

ACTION ACT_PeristalticPump_1:
fbRudongPumpModbusTcp[1].stPara.strSlaveIP:='192.168.1.60';
fbRudongPumpModbusTcp[1].stPara.nRemotePort:=1031;
fbRudongPumpModbusTcp[1].stPara.bySlaveID:=16#01;
//如果泵参数固定，就直接配置好，如果不固定，就在触摸屏配置
stData.RudongPump[1].iPumpType:=RudongPump_PumpType.DFPluse;//设定泵控制器类型
stData.RudongPump[1].iPumpTypeSet:=RudongPump_PumpHeadType.MiniPump01;//设定泵泵头类型
stData.RudongPump[1].iHosePipeTypeSet:=RudongPump_SoftPipeType.P19;//设定泵软管类型
FOR i:=1 TO gc_uiRudongPump DO
	fbRudongPumpModbusTcp[i].xAutoMode:=fbMachine[1].xAutoMode OR fbAutoCal.xRunning;
	fbRudongPumpModbusTcp[i](
	xExecute:= , 
	xAbort:= , 
	xResetRequest:=, 
	xRunILC:= true, 
	dwTimeLimit:= , 
	dwTimeOut:= , 
	stPara:= , 
	xNeedConfigurePara:= , 
	stRunPara:=stData.RudongPump[i] , 
	xAutoMode:= , 
	xIniting:= , 
	xDeviceRunning:= , 
	rSpeedRatio:= , 
	sHmiError:= , 
	xEStop:=fbMachine[1].xEStop or true , 
	stDeviceOpe:= , 
	xDone=> , 
	xBusy=> , 
	xError=> , 
	xAborted=> , 
	xRunning=> , 
	xRudongPump_ERROR=> , 
	eERRORID=> , 
	xRdyCmd=> );
END_FOR
END_ACTION

ACTION ACT_Proface:

fbProface[1](
	xEStop									:=fbMachine[1].xEStop,
	xSafety									:=fbMachine[1].xSafety,
	xManualMode							:=fbMachine[1].xManualMode,
	xAutoMode								:=fbMachine[1].xAutoMode,
	xAlarm									:=fbMachine[1].xAlarm,
	xTip										:=fbMachine[1].xTip,
	xInit										:=fbMachine[1].xInit,
	xIniting								:=fbMachine[1].xIniting,
	xInitDone								:=fbMachine[1].xInitDone,
	xDummyCheckDone					:=fbMachine[1].xDummyDone,
	xEmptyDone							:=fbMachine[1].xEmptyDone,
);
(*fbProface[1].strSystemTime[1]:=stDateTime.sTempTimeYYMMDD;
fbProface[1].strSystemTime[2]:=CONCAT(CONCAT( CONCAT(CONCAT(stDateTime.sTempTimeHO,':'),stDateTime.sTempTimeMI ),':'),stDateTime.sTempTimeSe);
*)
END_ACTION

ACTION ACT_Recipe:
(*FOR  iRec:=1 TO gc_RecipeNum BY 1 DO
	fb_Recipes[iRec](
	xICreateRecipe:= , 
	xILoadRecipe:= , 
	xIDeleteRecipe:= , 
	strRecipeDefinitionName:= , 
	RecipeName:= , 
	FileName:= , 
	xQBusy=> , 
	xQErrorID=> );
END_FOR
(************************Axis Recipe*************************)
fb_Recipes[1].strRecipeDefinitionName:='Recipe_Axis';
fb_Recipes[1].RecipeName:='Axis_1';
fb_Recipes[1].FileName:='\Hard Disk1\Recipefiles';
(************************Cylinder Recipe*************************)
fb_Recipes[2].strRecipeDefinitionName:='Recipe_Cylinder';
fb_Recipes[2].RecipeName:='Cylinder_1';
fb_Recipes[2].FileName:='\Hard Disk1\Recipefiles';
(************************RGI Recipe*************************)
fb_Recipes[3].strRecipeDefinitionName:='Recipe_RGI';
fb_Recipes[3].RecipeName:='RGI_1';
fb_Recipes[3].FileName:='\Hard Disk1\Recipefiles';
(************************Robot Recipe*************************)
fb_Recipes[4].strRecipeDefinitionName:='Recipe_Robot';
fb_Recipes[4].RecipeName:='Robot_1';
fb_Recipes[4].FileName:='\Hard Disk1\Recipefiles';
(************************Tray Recipe*************************)
fb_Recipes[5].strRecipeDefinitionName:='Recipe_Tray';
fb_Recipes[5].RecipeName:='Tray_1';
fb_Recipes[5].FileName:='\Hard Disk1\Recipefiles';
*)
END_ACTION

ACTION ACT_RGI_14:

	
IF NOT xRGI4_First THEN
	fbRGI_14_Modbus[1].stPara.bySlaveID := 1;
	fbRGI_14_Modbus[1].stPara.strSlaveIP := '192.168.1.90';//从站IP地址
	fbRGI_14_Modbus[1].stPara.iSlavePort := 1030;	
	xRGI4_First := TRUE;
ELSE
	//进行函数调用
	FOR i:=1 TO gc_uiRGI_14_Number BY 1 DO 
		fbRGI_14_Modbus[i](
		xExecute:= , 
		xAbort:=FALSE , 
		xPowerHmi:= TRUE, 
		xResetRequest:=fbMachine[1].xReset , 
		dwTimeLimit:= , 
		dwTimeOut:= , 
		stPara:= , 
		xAutoMode:=fbMachine[1].xAutoMode, 
		xIniting:= , 
		stPosPara:= stData.RGI14[i], 
		xDeviceRunning:= , 
		stOper:= , 
		xDone=> , 
		xBusy=> , 
		xAborted=> , 
		xError=> , 
		eErrorID=> , 
		xRdyCmd=> , 
		xRefOk=> , 
		eClampActCmd=> , 
		iClampStatus=> , 
		xGripClampEmpty=> , 
		xDropOccur=> , 
		xClosecoverFailure=> , 
		xOpencoverFailure=> , 
		sHmiError=> , 
		stRGIStates=> , 
		eCommErrorID=> , 
		eOperErrorID=> , 
		st_IOData:= st_RGI_IOData);
	END_FOR
END_IF


//手动输入初始值
IF xRecipeRGI14ParSetButton THEN 
	FOR i:=1 TO gc_uiRGI_14_Number BY 1 DO 
		FOR j:= 1 TO 5 BY 1 DO
			stData.RGI14[i].aHMIClampiPosAngleSet[j] := 
			stData.RGI14[i].aHMIClampiSpeedSet[j] := 
			stData.RGI14[i].aHMIClampiTorqueSet[j] := 
			stData.RGI14[i].aHMIReleasepiPosAngleSet[j] :=
			stData.RGI14[i].aHMIReleasepiSpeedSet[j]:= 
			stData.RGI14[i].aHMIReleasepiTorqueSet[j]:= 
			stData.RGI14[i].aHMIRotateClampiPosAngleSet[j] :=
			stData.RGI14[i].aHMIRotateClampiSpeedSet[j] :=
			stData.RGI14[i].aHMIRotateiTorqueSet[j] :=
			stData.RGI14[i].aHMIRotateReleaseiPosAngleSet[j] :=
			stData.RGI14[i].aHMIRotateReleaseiSpeedSet[j] :=
			stData.RGI14[i].aHMIRotateReleaseiTorqueSet[j]:= 100 ; 
	   END_FOR
	END_FOR
		xRecipeRGI14ParSetButton := FALSE ;
END_IF
END_ACTION

ACTION ACT_SmcVacuum:

FOR   i:=1 TO gc_uiValveNum BY 1 DO
 fbSmcVacuum[i](
	 xIAutoMode:=fbMachine[1].xAutoMode , 
	 xIManualMode:=fbMachine[1].xManualMode , 
	 xIVacuumWork:= , 
	 xIVacuumBroken:= , 
	 xIVacuumWorkHMI:= , 
	 xIVacuumBrokenHMI:= , 
	 xIDeviceRunning:= , 
	 xIVacuumWorkReached:= , 
	 xIVacuumBrokenReached:= , 
	 xQVacuumFeedValve=> , 
	 xQVacuumBrokenValve=> );
END_FOR

//真空吸反馈信号
fbSmcVacuum[1].xIVacuumWorkReached:=	IxS08Vacuum1_Output2	;//	卡片搬运工位¶真空发生器1¶输出OUT1
fbSmcVacuum[1].xIVacuumBrokenReached:=IxS08Vacuum1_Output1;//	卡片搬运工位¶真空发生器1¶输出OUT2
fbSmcVacuum[2].xIVacuumWorkReached:=IxS08Vacuum2_Output2	;//	卡片搬运工位¶真空发生器2¶输出OUT1
fbSmcVacuum[2].xIVacuumBrokenReached:=IxS08Vacuum2_Output1	;//	卡片搬运工位¶真空发生器2¶输出OUT2
//真空吸输出信号

QxVacuum1_FeedValveControl:=fbSmcVacuum[1].xQVacuumFeedValve;
QxVacuum1_BreakValveControl:=fbSmcVacuum[1].xQVacuumBrokenValve;
QxVacuum2_FeedValveControl:=fbSmcVacuum[2].xQVacuumFeedValve;
QxVacuum2_BreakValveControl:=fbSmcVacuum[2].xQVacuumBrokenValve;
END_ACTION

ACTION ACT_Station:
//上电复位
IF NOT xStation_First THEN
  FOR i:=1 TO gc_uiStationNum DO 
    fbStation[i].xCycleRunHmi:=FALSE;
    fbStation[i].xInitHmi:=FALSE;
    fbStation[i].xJogRunHmi:=FALSE;
    fbStation[i].xPauseHmi:=FALSE;
  END_FOR
  	xStation_First:=TRUE;
END_IF

FOR i:=1 TO gc_uiStationNum DO
	fbStation[i](
		xEStop:=fbMachine[1].xEStop , 
		xKey:=fbMachine[1].xKey , 
		xSafety:=fbMachine[1].xSafety , 
		xManualMode:=fbMachine[1].xManualMode , 
		xReset:=fbMachine[1].xReset , 
		xMachinePause:=fbMachine[1].xPause , 
		xMachineReInit:=fbMachine[1].xReInit , 
		xMachineIniting:=fbMachine[1].xIniting , 
		xMachineRunning:=fbMachine[1].xRunning , 
		tInitTimeout:= , 
		xInitHmi:= , 
		xInitDone:= , 
		xDisabled:= , 
		xCycleRunHmi:= , 
		xJogRunHmi:= , 
		xPauseHmi:= , 
		xCycleRunning=> , 
		xJogRunning=> , 
		xSingleRunning=> , 
		xRunning=> , 
		uiState=> , 
		diCycleTime =>   
	);
	StepAutoTransR_TRIG[i](CLK:=fbstation[i].xQStepAutoTrans , Q=> );
	IF StepAutoTransR_TRIG[i].Q  THEN
		FOR infor := 1 TO gc_StepHistory DO
			MEMCPY ( ADR(arStepAuto.Staion[i].History[infor-1]), ADR(arStepAuto.Staion[i].History[infor]), SIZEOF(arStepAuto.Staion[i].History[infor]));(* length      *)
		END_FOR		
		StepAutoTransR_TRIG[i](CLK:=FALSE );						
	END_IF
	
	 arStepAuto.Staion[i].History[gc_StepHistory]:=CONCAT(CONCAT(CONCAT('AutoStep:=' ,INT_TO_STRING(fbstation[i].iStepAuto)),'\\'),strLocalDateTime);
	 
	 
	 StepInitTransR_TRIG[i](CLK:=fbstation[i].xQStepInitTrans , Q=> );
	IF  StepInitTransR_TRIG[i].Q  THEN
		FOR infor := 1 TO gc_StepHistory DO
			MEMCPY ( ADR(arStepinit.Staion[i].History[infor-1]), ADR(arStepinit.Staion[i].History[infor]), SIZEOF(arStepinit.Staion[i].History[infor]));(* length      *)
		END_FOR	
		StepInitTransR_TRIG[i](CLK:=FALSE );										
	END_IF
	
	 	 arStepinit.Staion[i].History[gc_StepHistory]:=CONCAT(CONCAT(CONCAT('InitStep:=' ,INT_TO_STRING(fbstation[i].iStepInit)),'\\'),strLocalDateTime);
END_FOR
END_ACTION

ACTION ACT_System:

//	生成特定周期的振荡矩形波，可用于指示灯的闪烁，不可用于精确计时
fb_Blinker[1](
	tBlink:=T#10MS,
	bBlink=>stSysPulse.xP10ms,
	brBlink=>stSysPulse.xR10ms,
	bfBlink=>stSysPulse.xF10ms
);
fb_Blinker[2](
	tBlink:=T#20MS,
	bBlink=>stSysPulse.xP20ms,
	brBlink=>stSysPulse.xR20ms,
	bfBlink=>stSysPulse.xF20ms
);
fb_Blinker[3](
	tBlink:=T#50MS,
	bBlink=>stSysPulse.xP50ms,
	brBlink=>stSysPulse.xR50ms,
	bfBlink=>stSysPulse.xF50ms
);
fb_Blinker[4](
	tBlink:=T#100MS,
	bBlink=>stSysPulse.xP100ms,
	brBlink=>stSysPulse.xR100ms,
	bfBlink=>stSysPulse.xF100ms
);
fb_Blinker[5](
	tBlink:=T#200MS,
	bBlink=>stSysPulse.xP200ms,
	brBlink=>stSysPulse.xR200ms,
	bfBlink=>stSysPulse.xF200ms
);
fb_Blinker[6](
	tBlink:=T#500MS,
	bBlink=>stSysPulse.xP500ms,
	brBlink=>stSysPulse.xR500ms,
	bfBlink=>stSysPulse.xF500ms
);
fb_Blinker[7](
	tBlink:=T#1S,
	bBlink=>stSysPulse.xP1s,
	brBlink=>stSysPulse.xR1s,
	bfBlink=>stSysPulse.xF1s
);
fb_Blinker[8](
	tBlink:=T#2S,
	bBlink=>stSysPulse.xP2s,
	brBlink=>stSysPulse.xR2s,
	bfBlink=>stSysPulse.xF2s
);
fb_Blinker[9](
	tBlink:=T#5S,
	bBlink=>stSysPulse.xP5s,
	brBlink=>stSysPulse.xR5s,
	bfBlink=>stSysPulse.xF5s
);
fb_Blinker[10](
	tBlink:=T#10S,
	bBlink=>stSysPulse.xP10s,
	brBlink=>stSysPulse.xR10s,
	bfBlink=>stSysPulse.xF10s
);
END_ACTION

ACTION ACT_TURINRobot:
IF NOT _firstTURINRobot
THEN
	fbTURINContorl[1].stPara.strSlaveIP := '192.168.1.111';
	fbTURINContorl[1].stPara.bySlaveID := 1;
	fbTURINContorl[1].stPara.iSlavePort :=502;
	_firstTURINRobot := TRUE;
ELSE
	//控制功能块实例化
	FOR i:=1 TO gc_uiTURINRobot_Num DO
		fbTURINContorl[i](
			xManuMode:= fbMachine[1].xManualMode , 
			xAutoRunning:= fbMachine[1].xRunning , 
			xEStop:= fbMachine[1].xEStop  ,  
			xReset:= (fbMachine[1].xReset ) , 
			xStart:= (fbMachine[1].xStart ) , 
			xStop:= fbMachine[1].xStop , 
			xPause:= fbMachine[1].xPause , 
			xMovePermit:=  fbStation[7].xAlarm AND  NOT  fbMachine[1].xSafety AND stFromRobot.xLocal_Remote,
			xContinue:= , 
			//xInitExte:= S03_Robot.xInit, 
			xInitExte:=,
			xClearInitedFlag:= , 
			xInitedFlag=> , 
			xInitFinish=> , 
			iCurrentStatus=> , 
			eErrID=> ,
      stData:=stData.TURIN[i]);	

    END_FOR	


END_IF
//TO ROBOT
fbTURINContorl[1].pSysToRobot[1]    := stToRobot1.iMoveMode; 
fbTURINContorl[1].pSysToRobot[2]    := stToRobot1.iRatio;
fbTURINContorl[1].pSysToRobot[3].0  := stToRobot1.xStepRunPermit;
fbTURINContorl[1].pSysToRobot[3].1  := stToRobot1.xPickPos1Premit ;      
fbTURINContorl[1].pSysToRobot[3].2  := stToRobot1.xPickPos2Premit  ;      
fbTURINContorl[1].pSysToRobot[3].3  := stToRobot1.xPickPos3Premit ;       
fbTURINContorl[1].pSysToRobot[3].4  := stToRobot1.xPickTransferPosPremit; 
fbTURINContorl[1].pSysToRobot[3].5  := stToRobot1.xPutPos1Premit    ;     
fbTURINContorl[1].pSysToRobot[3].6  := stToRobot1.xPutPos2Premit    ;     
fbTURINContorl[1].pSysToRobot[3].7  := stToRobot1.xPutPos3Premit    ;    
fbTURINContorl[1].pSysToRobot[3].8  := stToRobot1.xPutPos4Premit    ;     
fbTURINContorl[1].pSysToRobot[3].9  := stToRobot1.xClampPartDone  ;     
fbTURINContorl[1].pSysToRobot[3].10 := stToRobot1.xReleasePartDone ;    

//FROM ROBOT
stFromRobot.xEstop					  	    := fbTURINContorl[1].pSysFromRobot[0].00;
stFromRobot.xLocal_Remote				    := fbTURINContorl[1].pSysFromRobot[0].02;
stFromRobot.xEnable				          := fbTURINContorl[1].pSysFromRobot[0].03;
stFromRobot.xRuntip				          := fbTURINContorl[1].pSysFromRobot[1].08;
stFromRobot.xStopTip				        := fbTURINContorl[1].pSysFromRobot[1].09;
                                    
stFromRobot1.xHomePosReached         	 	 := fbTURINContorl[1].pSysFromRobot[3].00;
stFromRobot1.xPickPos1Reached              := fbTURINContorl[1].pSysFromRobot[3].01;
stFromRobot1.xPickPos2Reached              := fbTURINContorl[1].pSysFromRobot[3].02;
stFromRobot1.xPickPos3Reached              := fbTURINContorl[1].pSysFromRobot[3].03;
stFromRobot1.xPickTransferPosReached       := fbTURINContorl[1].pSysFromRobot[3].04;
stFromRobot1.xPutPos1Reached          	    := fbTURINContorl[1].pSysFromRobot[3].05;
stFromRobot1.xPutPos2Reached               := fbTURINContorl[1].pSysFromRobot[3].06;
stFromRobot1.xPutPos3Reached         	    := fbTURINContorl[1].pSysFromRobot[3].07;
stFromRobot1.xPutPos4Reached          	    := fbTURINContorl[1].pSysFromRobot[3].08;
stFromRobot1.xStepRunning                  := fbTURINContorl[1].pSysFromRobot[3].09;
stFromRobot1.xStepRunDone                  := fbTURINContorl[1].pSysFromRobot[3].10;
stFromRobot1.xInitOK                      	:= fbTURINContorl[1].pSysFromRobot[3].11;
stFromRobot1.xOutofseg1                     := fbTURINContorl[1].pSysFromRobot[3].14;
stFromRobot1.xOutofseg2                     := fbTURINContorl[1].pSysFromRobot[3].12;
stFromRobot1.xOutofseg3                     := fbTURINContorl[1].pSysFromRobot[3].13;
END_ACTION

ACTION ACT_UPS:
GVL_UPS.fb_1sUPS(
	sNetID:= , 
	iPLCPort:=851 , 
	iUPSPort:=16#588 , 
	tTimeout:= , 
	eUpsMode:=eSUPS_WrPersistData_Shutdown , 
	ePersistentMode:=SPDM_2PASS , 
	tRecoverTime:=T#20S , 
	bPowerFailDetect=> , 
	eState=> );
	
IF  eGlobalSUpsState =eSUPS_PowerOK    THEN  ///外部供电正常  
	///写程序
ELSIF   eGlobalSUpsState = eSUPS_PowerFailure THEN//外部断电（这种状态只会持续1个PLC周期）
	
	///写程序
ELSIF   eGlobalSUpsState  =   eSUPS_WritePersistentData THEN  //在写掉电保持参数，（详见第八章讲叙的UPS断电和启动过程）
	
	///写程序
ELSIF       eGlobalSUpsState  =   eSUPS_QuickShutdown   THEN  //系统开始快速关机
	///写程序
	
ELSIF    eGlobalSUpsState  =   eSUPS_WaitForRecover     THEN//等待外部供电恢复
	///写程序

ELSIF    eGlobalSUpsState  =  eSUPS_WaitForPowerOFF     THEN//等待UPS电量耗尽关机
	///写程序

END_IF
END_ACTION

ACTION ACT_WritePersistentData:
//写入保持性存储区

fbWritePersistentData(
	NETID:= '', 
	PORT:= 851, 
	START:= stSysPulse.xP5s , 
	TMOUT:= , 
	MODE:= , 
	BUSY=> , 
	ERR=> , 
	ERRID=> );
END_ACTION

ACTION ACT_Z_ERG_20:

	fbERG_20_Modbus[1].stPara.bySlaveID := 1;
	fbERG_20_Modbus[1].stPara.strSlaveIP := '192.168.1.20';//从站IP地址
	fbERG_20_Modbus[1].stPara.iSlavePort := 1030;	//四端口智嵌物联
	
	fbERG_20_Modbus[2].stPara.bySlaveID := 1;
	fbERG_20_Modbus[2].stPara.strSlaveIP := '192.168.1.21';//从站IP地址
	fbERG_20_Modbus[2].stPara.iSlavePort := 1031;
	//进行函数调用
FOR i := 1 TO gc_uiHITBOT_Number BY 1 DO
fbERG_20_Modbus[i](
	xExecute:= , 
	xAbort:= , 
	xResetRequest:=fbMachine[1].xReset , 
	xPowerHmi:=TRUE , 
	dwTimeLimit:= , 
	dwTimeOut:= , 
	stPara:= , 
	xHMInitButton:= , 
	xInitControl:= , 
	aHMIClampButton:= , 
	aHMIReleaseButton:= , 
	aClampControl:= , 
	aReleaseControl:= , 
	aHMIRotateClampButton:= , 
	aHMIRotateReleaseButton:= , 
	aRotateClampControl:= , 
	aRotateReleaseControl:= , 
	aHMIRotateClampRelButton:= , 
	aHMIRotateReleaseRelButton:= , 
	aRotateClampRelControl:= , 
	aRotateReleaseRelControl:= , 
	aHMIClampPara:=stData.ERG20[i].aHMIClampPara , 
	aHMIReleasePara:=stData.ERG20[i].aHMIReleasePara , 
	aHMIRotateClampPara:=stData.ERG20[i].aHMIRotateClampPara , 
	aHMIRotateReleasePara:=stData.ERG20[i].aHMIRotateReleasePara , 
	aHMIRotateClampRelPara:=stData.ERG20[i].aHMIRotateRelClampPara , 
	aHMIRotateReleaseRelPara:=stData.ERG20[i].aHMIRotateRelReleasePara , 
	xAutoMode:= fbMachine[1].xAutoMode, 
	xDeviceRunning:= , 
	xDone=> , 
	xBusy=> , 
	xAborted=> , 
	xError=> , 
	eErrorID=> , 
	xRdyCmd=> , 
	xRefOk=> , 
	xGripClampEmpty=> , 
	xDropOccur=> , 
	sHmiError=> , 
	eCommErrorID=> , 
	eOperErrorID=> , 
	st_IOData:= stZ_ERG_20_IOData[i] );
END_FOR
END_ACTION

END_PROGRAM

// ---- POUs/003_FB/41_GetSystemTime/PRG_GetSystemTime.TcPOU
PROGRAM PRG_GetSystemTime
VAR_OUTPUT
	sQTime:	TIMESTRUCT;	(* Output: Timeinformation *)
END_VAR
VAR
	fbNTGetTime:	NT_GetTime;
	fbTONGetTime:	TON;
END_VAR


(* Receive the NT-Time every second *)
fbTONGetTime( IN := TRUE, PT := T#1s );
IF fbTONGetTime.Q THEN
	fbNTGetTime( START := FALSE );
	fbTONGetTime( IN := FALSE );
END_IF
fbNTGetTime
	(	START := TRUE,
		TMOUT := DEFAULT_ADS_TIMEOUT
	);

(* Setting the result *)
sQTime	:= fbNTGetTime.TIMESTR;

END_PROGRAM

// ---- POUs/002_Machine/CommWithPC.TcPOU
PROGRAM CommWithPC
VAR
END_VAR

ACT_Send();

ACTION ACT_Receive:
//1.iPCALive	:INT	;//	心跳	保持1s跳动为正常，否则5s为异常

//2.打打印机准备就绪
//	 iLableReady	:INT	;//	打印机贴标准备就绪	1=准备就绪  0=未就绪
//	 iMachineLampButton	:INT	;//	设备灯控制	1=开灯，0=关灯
//	 iInitComfirm	:INT	;//		1=初始化确认  
//	 iShiftButton	:INT	;//	订单下发按钮	1=订单下发
//	 iMachineEmptyButton	:INT	;//	设备清空按钮	1=设备清空
//	 iPCAlarm	:INT	;//	PC报警	1=有报警   0 =无报警
//	 iBodyType	:INT	;//	设备产品类型	1…n:分别代表的产品类型
//	 iScrapLabel	:INT	;//	废弃空白标签	0=不废弃    1= 废弃空白标签
//	 iShiftTotal	:INT	;//	订单总数	订单总数下发
//	 iEmptyButtonComfirm:INT;//设备清空确认
END_ACTION

ACTION ACT_Send:
//1.心跳见ACT_ALIVE
//2.清空完成信号
IF  fbMachine[1].xEmptyDone THEN
		sPLC_TO_PC.iMachineEmptyDone:=1;
ELSE
 		sPLC_TO_PC.iMachineEmptyDone:=0;
END_IF
//3.贴标完成
	IF  S13_Labeling.xQLabelCompleted THEN
			sPLC_TO_PC.iLableCompeted:=1;
	ELSE
	 			sPLC_TO_PC.iLableCompeted:=0;
	END_IF
//4.设备初始化命令
	IF  fbMachine[1].xInit THEN
			sPLC_TO_PC.iInitCommand:=1;
	END_IF
//5.初始化完成命令
	 IF   fbMachine[1].xInitDone THEN
			sPLC_TO_PC.iInitFinished:=1;
		END_IF
//6.设备启动
	 IF   fbMachine[1].xStart THEN
			 sPLC_TO_PC.iMachineStart:=1;
		END_IF

//7.	iShiftOKTotal	:INT;		//	订单OK件计数		
//8.	iShiftNGTotal	:INT;		//	订单NG件计数	

//9.	iRobotUnloadSignal:INT	;//机械手下料信号	1=机械手下料完成   用于计算设备CT
END_ACTION

END_PROGRAM

// ---- POUs/001_Station/001_Mapping/OutputLink.TcPOU
PROGRAM OutputLink
VAR
END_VAR

ACT_ET01();
ACT_ET02();
ACT_ET03();
ACT_ET04();

ACTION ACT_ET01:
ET01_Output[1].Output.0	:=	QxStartButtonLamp	;//	启动按钮指示灯
ET01_Output[1].Output.1	:=	QxStopButtonLamp	;//	停止按钮指示灯
ET01_Output[1].Output.2	:=	QxResetButtonLamp	;//	复位按钮指示灯
ET01_Output[1].Output.3	:=	QxInitButtonLamp	;//	初始化按钮指示灯
ET01_Output[1].Output.4	:=	QxIonStopControl	;//	上料工位¶离子风棒¶停止放电信号
ET01_Output[1].Output.5	:=	QxIonCheckDirtyControl	;//	上料工位¶离子风棒¶电极针脏污检出信号
ET01_Output[1].Output.6	:=	QxFlowLineStart	;//	链板线电机¶正转输出
ET01_Output[1].Output.7	:=	QxFlowLineStop	;//	链板线电机¶停止输出
ET01_Output[1].Output.8	:=	QxFlowLineSpeedCtrl_1	;//	链板线电机¶多段速1输出
ET01_Output[1].Output.9	:=	QxFlowLineSpeedCtrl_2	;//	链板线电机¶多段速2输出
ET01_Output[1].Output.10	:=	QxMachineLamp1Control	;//	日光灯1控制
ET01_Output[1].Output.11	:=	QxMachineLamp2Control	;//	日光灯2控制
ET01_Output[1].Output.12	:=	QxRedLamp	;//	三色灯-红灯
ET01_Output[1].Output.13	:=	QxYellowLamp	;//	三色灯-黄灯
ET01_Output[1].Output.14	:=	QxGreenLamp	;//	三色灯-绿灯
ET01_Output[1].Output.15	:=	QxBuzzer	;//	三色-蜂鸣器灯
ET01_Output[2].Output.0	:=	QxS01VTCPressCyl_1WP	;//	链板线¶Z轴阻挡气缸1¶动点输出
ET01_Output[2].Output.1	:=	QxS01VTCPressCyl_1HP	;//	链板线¶Z轴阻挡气缸1¶原点输出
ET01_Output[2].Output.2	:=	QxS01VTCPressCyl_2WP	;//	链板线¶Z轴阻挡气缸2¶动点输出
ET01_Output[2].Output.3	:=	QxS01VTCPressCyl_2HP	;//	链板线¶Z轴阻挡气缸2¶原点输出
ET01_Output[2].Output.4	:=	QxS01VTCPressCyl_3WP	;//	链板线¶Z轴阻挡气缸3¶动点输出
ET01_Output[2].Output.5	:=	QxS01VTCPressCyl_3HP	;//	链板线¶Z轴阻挡气缸3¶原点输出
ET01_Output[2].Output.6	:=	QxS01VTCPressCyl_4WP	;//	链板线¶Z轴阻挡气缸4¶动点输出
ET01_Output[2].Output.7	:=	QxS01VTCPressCyl_4HP	;//	链板线¶Z轴阻挡气缸4¶原点输出
ET01_Output[2].Output.8	:=	QxS01VTCCyl_1WP	;//	上料工位¶移栽Z轴气缸1¶动点输出
ET01_Output[2].Output.9	:=	QxS01VTCCyl_1HP	;//	上料工位¶移栽Z轴气缸¶原点输出
ET01_Output[2].Output.10	:=	QxS01VTCCyl_2WP	;//	上料工位¶移栽Z轴气缸2¶动点输出
ET01_Output[2].Output.11	:=	QxS01VTCCyl_2HP	;//	上料工位¶移栽变距气缸¶原点输出
ET01_Output[2].Output.12	:=	QxS02HOZAdjustCyl_1WP	;//	注液工位¶上层水平调整气缸1¶动点输出
ET01_Output[2].Output.13	:=	QxS02HOZAdjustCyl_1HP	;//	注液工位¶上层水平调整气缸1¶原点输出
ET01_Output[2].Output.14	:=	QxShare40	;//	备用
ET01_Output[2].Output.15	:=	QxShare41	;//	备用
ET01_Output[3].Output.0	:=	QxS02HOZAdjustCyl_3WP	;//	注液工位¶下层水平调整气缸1¶动点输出
ET01_Output[3].Output.1	:=	QxS02HOZAdjustCyl_3HP	;//	注液工位¶下层水平调整气缸1¶原点输出
ET01_Output[3].Output.2	:=	QxShare42	;//	备用
ET01_Output[3].Output.3	:=	QxShare43	;//	备用
ET01_Output[3].Output.4	:=	QxS02ROTCylWP	;//	注液工位¶防滴液¶动点输出
ET01_Output[3].Output.5	:=	QxS02ROTCylHP	;//	注液工位¶防滴液¶原点输出
ET01_Output[3].Output.6	:=	QxS03HOZAdjustCyl_1WP	;//	相机工位¶上层水平调整气缸1¶动点输出
ET01_Output[3].Output.7	:=	QxS03HOZAdjustCyl_1HP	;//	相机工位¶上层水平调整气缸1¶原点输出
ET01_Output[3].Output.8	:=	QxS03HOZAdjustCyl_2WP	;//	相机工位¶上层水平调整气缸2¶动点输出
ET01_Output[3].Output.9	:=	QxS03HOZAdjustCyl_2HP	;//	相机工位¶上层水平调整气缸2¶原点输出
ET01_Output[3].Output.10	:=	QxS03HOZAdjustCyl_3WP	;//	相机工位¶上层水平调整气缸3¶动点输出
ET01_Output[3].Output.11	:=	QxS03HOZAdjustCyl_3HP	;//	相机工位¶上层水平调整气缸3¶原点输出
ET01_Output[3].Output.12	:=	QxS03HOZAdjustCyl_4WP	;//	相机工位¶上层水平调整气缸4¶动点输出
ET01_Output[3].Output.13	:=	QxS03HOZAdjustCyl_4HP	;//	相机工位¶上层水平调整气缸4¶原点输出
ET01_Output[3].Output.14	:=	QxS03HOZAdjustCyl_5WP	;//	相机工位¶上层水平调整气缸5¶动点输出
ET01_Output[3].Output.15	:=	QxS03HOZAdjustCyl_5HP	;//	相机工位¶上层水平调整气缸5¶原点输出
ET01_Output[4].Output.0	:=	QxS03HOZAdjustCyl_6WP	;//	相机工位¶上层水平调整气缸6¶动点输出
ET01_Output[4].Output.1	:=	QxS03HOZAdjustCyl_6HP	;//	相机工位¶上层水平调整气缸6¶原点输出
ET01_Output[4].Output.2	:=	QxS03HOZAdjustCyl_7WP	;//	相机工位¶上层水平调整气缸7¶动点输出
ET01_Output[4].Output.3	:=	QxS03HOZAdjustCyl_7HP	;//	相机工位¶上层水平调整气缸7¶原点输出
ET01_Output[4].Output.4	:=	QxS03HOZAdjustCyl_8WP	;//	相机工位¶上层水平调整气缸8¶动点输出
ET01_Output[4].Output.5	:=	QxS03HOZAdjustCyl_8HP	;//	相机工位¶上层水平调整气缸8¶原点输出
ET01_Output[4].Output.6	:=	QxS04AluCoverCylWP	;//	铝膜胀气轴
ET01_Output[4].Output.7	:=	QxShare8	;//	备用
ET01_Output[4].Output.8	:=	QxShare9	;//	备用
ET01_Output[4].Output.9	:=	QxShare10	;//	备用
ET01_Output[4].Output.10	:=	QxShare11	;//	备用
ET01_Output[4].Output.11	:=	QxShare12	;//	备用
ET01_Output[4].Output.12	:=	QxShare13	;//	备用
ET01_Output[4].Output.13	:=	QxShare14	;//	备用
ET01_Output[4].Output.14	:=	QxShare15	;//	备用
ET01_Output[4].Output.15	:=	QxShare16	;//	备用
ET01_Output[5].Output.0	:=	QxCamera1Trigger	;//	相机检测工位¶相机触发1
ET01_Output[5].Output.1	:=	QxCamera2Trigger	;//	相机检测工位¶相机触发2
ET01_Output[5].Output.2	:=	QxCamera3Trigger	;//	相机检测工位¶相机触发3
ET01_Output[5].Output.3	:=	QxCamera4Trigger	;//	相机检测工位¶相机触发4
ET01_Output[5].Output.4	:=	QxCamera5Trigger	;//	相机检测工位¶相机触发5
ET01_Output[5].Output.5	:=	QxCamera6Trigger	;//	相机检测工位¶相机触发6
ET01_Output[5].Output.6	:=	QxCamera7Trigger	;//	相机检测工位¶相机触发7
ET01_Output[5].Output.7	:=	QxCamera8Trigger	;//	相机检测工位¶相机触发8
ET01_Output[5].Output.8	:=	QxCamera9Trigger	;//	相机检测工位¶相机触发9
ET01_Output[5].Output.9	:=	QxCamera10Trigger	;//	相机检测工位¶相机触发10
ET01_Output[5].Output.10	:=	QxCamera11Trigger	;//	相机检测工位¶相机触发11
ET01_Output[5].Output.11	:=	QxCamera12Trigger	;//	相机检测工位¶相机触发12
ET01_Output[5].Output.12	:=	QxCamera13Trigger	;//	相机检测工位¶相机触发13
ET01_Output[5].Output.13	:=	QxCamera14Trigger	;//	相机检测工位¶相机触发14
ET01_Output[5].Output.14	:=	QxCamera15Trigger	;//	相机检测工位¶相机触发15
ET01_Output[5].Output.15	:=	QxCamera16Trigger	;//	相机检测工位¶相机触发16
ET01_Output[6].Output.0	:=	QxCamera17Trigger	;//	相机检测工位¶相机触发17
ET01_Output[6].Output.1	:=	QxCameraLight1Trigger	;//	相机光源触发通道1
ET01_Output[6].Output.2	:=	QxCameraLight2Trigger	;//	相机光源触发通道2
ET01_Output[6].Output.3	:=	QxCameraLight3Trigger	;//	相机光源触发通道3
ET01_Output[6].Output.4	:=	QxCameraLight4Trigger	;//	相机光源触发通道4
ET01_Output[6].Output.5	:=	QxShare21	;//	备用
ET01_Output[6].Output.6	:=	QxShare22	;//	备用
ET01_Output[6].Output.7	:=	QxShare23	;//	备用
ET01_Output[6].Output.8	:=	QxShare24	;//	备用
ET01_Output[6].Output.9	:=	QxShare25	;//	备用
ET01_Output[6].Output.10	:=	QxShare26	;//	备用
ET01_Output[6].Output.11	:=	QxShare27	;//	备用
ET01_Output[6].Output.12	:=	QxShare28	;//	备用
ET01_Output[6].Output.13	:=	QxShare29	;//	备用
ET01_Output[6].Output.14	:=	QxShare30	;//	备用
ET01_Output[6].Output.15	:=	QxShare31	;//	备用
END_ACTION

ACTION ACT_ET02:
ET02_Output[1].Output.0	:=	QxRedLamp_1	;//	三色灯-红灯
ET02_Output[1].Output.1	:=	QxYellowLamp_1	;//	三色灯-黄灯
ET02_Output[1].Output.2	:=	QxGreenLamp_1	;//	三色灯-绿灯
ET02_Output[1].Output.3	:=	QxBuzzer_1	;//	三色灯-蜂鸣器灯
ET02_Output[1].Output.4	:=	QxHeatRelayContorl1	;//	加热棒供电接触器1
ET02_Output[1].Output.5	:=	QxHeatRelayContorl2	;//	加热棒供电接触器2
ET02_Output[1].Output.6	:=	QxMachineLamp3Contorl	;//	日光灯控制
ET02_Output[1].Output.7	:=	QxVacuum1_FeedValveControl	;//	卡片搬运工位¶真空发生器1¶供给阀控制
ET02_Output[1].Output.8	:=	QxVacuum1_BreakValveControl	;//	卡片搬运工位¶真空发生器1¶破坏阀控制
ET02_Output[1].Output.9	:=	QxVacuum2_FeedValveControl	;//	卡片搬运工位¶真空发生器2¶供给阀控制
ET02_Output[1].Output.10	:=	QxVacuum2_BreakValveControl	;//	卡片搬运工位¶真空发生器2¶破坏阀控制
ET02_Output[1].Output.11	:=	QxET02IonControlSignal1	;//	卡片搬运工位¶离子风棒¶外部给定信号1
ET02_Output[1].Output.12	:=	QxET02IonControlSignal2	;//	卡片搬运工位¶离子风棒¶外部给定信号2
ET02_Output[1].Output.13	:=	QxET02IonStopControl	;//	卡片搬运工位¶离子风棒¶停止放电信号
ET02_Output[1].Output.14	:=	QxET02IonResetControl	;//	卡片搬运工位¶离子风棒¶复位信号
ET02_Output[1].Output.15	:=	QxS09ControlValve	;//	卡片搬运工位¶离子风棒¶电磁阀控制
ET02_Output[2].Output.0	:=	QxS04HOZAdjustCyl_1WP	;//	热熔工位¶上层水平调整气缸1¶动点输出
ET02_Output[2].Output.1	:=	QxS04HOZAdjustCyl_1HP	;//	热熔工位¶上层水平调整气缸1¶原点输出
ET02_Output[2].Output.2	:=	QxShare75	;//	备用
ET02_Output[2].Output.3	:=	QxShare76	;//	备用
ET02_Output[2].Output.4	:=	QxS04HOZAdjustCyl_3WP	;//	热熔工位¶下层水平调整气缸1¶动点输出
ET02_Output[2].Output.5	:=	QxS04HOZAdjustCyl_3HP	;//	热熔工位¶下层水平调整气缸1¶原点输出
ET02_Output[2].Output.6	:=	QxShare77	;//	备用
ET02_Output[2].Output.7	:=	QxShare78	;//	备用
ET02_Output[2].Output.8	:=	QxS06GlampCyl_1WP	;//	切膜工位¶前侧夹膜气缸¶动点输出
ET02_Output[2].Output.9	:=	QxS06GlampCyl_1HP	;//	切膜工位¶前侧夹膜气缸¶原点输出
ET02_Output[2].Output.10	:=	QxS06GlampCyl_2WP	;//	切膜工位¶后侧夹膜气缸¶动点输出
ET02_Output[2].Output.11	:=	QxS06GlampCyl_2HP	;//	切膜工位¶后侧夹膜气缸¶原点输出
ET02_Output[2].Output.12	:=	QxS06HOZReachedCyl_1WP	;//	切膜工位¶水平到位气缸1¶动点出输出
ET02_Output[2].Output.13	:=	QxS06HOZReachedCyl_1HP	;//	切膜工位¶水平到位气缸1¶原点出输出
ET02_Output[2].Output.14	:=	QxS06HOZReachedCyl_2WP	;//	切膜工位¶水平到位气缸2¶动点输出
ET02_Output[2].Output.15	:=	QxS06HOZReachedCyl_2HP	;//	切膜工位¶水平到位气缸2¶原点输出
ET02_Output[3].Output.0	:=	QxS06HOZCyl_1WP	;//	切膜工位¶水平切膜气缸¶动点输出
ET02_Output[3].Output.1	:=	QxS06HOZCyl_1HP	;//	切膜工位¶水平切膜气缸¶原点输出
ET02_Output[3].Output.2	:=	QxS06VTCAdjustCylWP	;//	切膜工位¶下方对中顶升气缸¶动点输出
ET02_Output[3].Output.3	:=	QxS06VTCAdjustCylHP	;//	切膜工位¶下方对中顶升气缸¶原点输出
ET02_Output[3].Output.4	:=	QxS06GlampAdjustCyl_1WP	;//	切膜工位¶下方对中夹爪气缸1¶动点输出
ET02_Output[3].Output.5	:=	QxS06GlampAdjustCyl_1HP	;//	切膜工位¶下方对中夹爪气缸1¶原点输出
ET02_Output[3].Output.6	:=	QxS06GlampAdjustCyl_2WP	;//	切膜工位¶下方对中夹爪气缸2¶动点输出
ET02_Output[3].Output.7	:=	QxS06GlampAdjustCyl_2HP	;//	切膜工位¶下方对中夹爪气缸2¶原点输出
ET02_Output[3].Output.8	:=	QxS06GlampAdjustCyl_3WP	;//	切膜工位¶下方对中夹爪气缸3¶动点输出
ET02_Output[3].Output.9	:=	QxS06GlampAdjustCyl_3HP	;//	切膜工位¶下方对中夹爪气缸3¶原点输出
ET02_Output[3].Output.10	:=	QxS08HOZCylWP	;//	卡片工位¶水平气缸¶动点输出
ET02_Output[3].Output.11	:=	QxS08HOZCylHP	;//	卡片工位¶水平气缸¶原点输出
ET02_Output[3].Output.12	:=	QxS08VTCCyl_1WP	;//	卡片工位¶Z轴气缸1¶动点输出
ET02_Output[3].Output.13	:=	QxS08VTCCyl_1HP	;//	卡片工位¶Z轴气缸1¶原点输出
ET02_Output[3].Output.14	:=	QxS08VTCCyl_2WP	;//	卡片工位¶Z轴气缸2¶动点输出
ET02_Output[3].Output.15	:=	QxS08VTCCyl_2HP	;//	卡片工位¶Z轴气缸2¶原点输出
ET02_Output[4].Output.0	:=	QxS06PressCyl_1WP	;//	切膜下压气缸1动点输出
ET02_Output[4].Output.1	:=	QxS06PressCyl_1HP	;//	切膜下压气缸1原点输出
ET02_Output[4].Output.2	:=	QxS06PressCyl_2WP	;//	切膜下压气缸2动点输出
ET02_Output[4].Output.3	:=	QxS06PressCyl_2HP	;//	切膜下压气缸2原点输出
ET02_Output[4].Output.4	:=	QxS06VTCCylWP	;//	垂直切膜气缸1动点输出
ET02_Output[4].Output.5	:=	QxS06VTCCylHP	;//	垂直切膜气缸2原点输出
ET02_Output[4].Output.6	:=	QxS06BlowValve	;//切膜工位铝膜吹气电磁阀
ET02_Output[4].Output.7	:=	QxShare87	;//	备用
ET02_Output[4].Output.8	:=	QxShare88	;//	备用
ET02_Output[4].Output.9	:=	QxShare89	;//	备用
ET02_Output[4].Output.10	:=	QxShare90	;//	备用
ET02_Output[4].Output.11	:=	QxShare91	;//	备用
ET02_Output[4].Output.12	:=	QxShare92	;//	备用
ET02_Output[4].Output.13	:=	QxShare93	;//	备用
ET02_Output[4].Output.14	:=	QxShare94	;//	备用
ET02_Output[4].Output.15	:=	QxShare95	;//	备用
END_ACTION

ACTION ACT_ET03:
ET03_Output[1].Output.0	:=	QxLoadCell_1ZeroInput	;//	压力传感器1清零信号
ET03_Output[1].Output.1	:=	QxLoadCell_2ZeroInput	;//	压力传感器2清零信号
ET03_Output[1].Output.2	:=	QxLoadCell_3ZeroInput	;//	压力传感器3清零信号
ET03_Output[1].Output.3	:=	QxLoadCell_4ZeroInput	;//	压力传感器4清零信号
ET03_Output[1].Output.4	:=	QxLoadCell_5ZeroInput	;//	压力传感器5清零信号
ET03_Output[1].Output.5	:=	QxLoadCell_6ZeroInput	;//	压力传感器6清零信号
ET03_Output[1].Output.6	:=	QxShare165	;//	备用
ET03_Output[1].Output.7	:=	QxShare166	;//	备用
ET03_Output[1].Output.8	:=	QxShare167	;//	备用
ET03_Output[1].Output.9	:=	QxShare168	;//	备用
ET03_Output[1].Output.10	:=	QxShare169	;//	备用
ET03_Output[1].Output.11	:=	QxShare170	;//	备用
ET03_Output[1].Output.12	:=	QxShare171	;//	备用
ET03_Output[1].Output.13	:=	QxShare172	;//	备用
ET03_Output[1].Output.14	:=	QxShare173	;//	备用
ET03_Output[1].Output.15	:=	QxShare174	;//	备用
END_ACTION

ACTION ACT_ET04:
ET04_Output[1].Output.0	:=	QxMotorForward	;//	热缩封膜出料线体¶电机正转
ET04_Output[1].Output.1	:=	QxMotorStop	;//	热缩封膜出料线体¶电机停止
ET04_Output[1].Output.2	:=	QxMotorBackward	;//	热缩封膜出料线体¶电机反转
ET04_Output[1].Output.3	:=	QxMotorReserve	;//	热缩封膜出料线体¶电机备用
ET04_Output[1].Output.4	:=	QxCameraTrigger	;//	相机触发
ET04_Output[1].Output.5	:=	QxLabelStart	;//	贴标机Start
ET04_Output[1].Output.6	:=	QxLabelRibwarn	;//	贴标机RIBWARN
ET04_Output[1].Output.7	:=	QxLabelReset	;//	贴标机RESET
ET04_Output[1].Output.8	:=	QxS11HOZCylWP	;//	贴标处推料气缸¶动点
ET04_Output[1].Output.9	:=	QxS11HOZCylHP	;//	贴标处推料气缸¶原点
ET04_Output[1].Output.10	:=	QxS12HOZCyl_1WP	;//	贴标检测工位¶推料气缸1¶动点
ET04_Output[1].Output.11	:=	QxS12HOZCyl_1HP	;//	贴标检测工位¶推料气缸1¶原点
ET04_Output[1].Output.12	:=	QxS12HOZCyl_2WP	;//	贴标检测工位¶推料气缸2¶动点
ET04_Output[1].Output.13	:=	QxS12HOZCyl_2HP	;//	贴标检测工位¶推料气缸2¶原点
ET04_Output[1].Output.14	:=	QxS13HOZCyl_1WP	;//	NG推料气缸1¶动点
ET04_Output[1].Output.15	:=	QxS13HOZCyl_1HP	;//	NG推料气缸1¶原点
ET04_Output[2].Output.0	:=	QxS13HOZCyl_2WP	;//	NG推料气缸2¶动点
ET04_Output[2].Output.1	:=	QxS13HOZCyl_2HP	;//	NG推料气缸2¶原点
ET04_Output[2].Output.2	:=	QxShare150	;//	备用
ET04_Output[2].Output.3	:=	QxShare151	;//	备用
ET04_Output[2].Output.4	:=	QxShare152	;//	备用
ET04_Output[2].Output.5	:=	QxShare153	;//	备用
ET04_Output[2].Output.6	:=	QxShare154	;//	备用
ET04_Output[2].Output.7	:=	QxShare155	;//	备用
ET04_Output[2].Output.8	:=	QxShare156	;//	备用
ET04_Output[2].Output.9	:=	QxShare157	;//	备用
ET04_Output[2].Output.10	:=	QxShare158	;//	备用
ET04_Output[2].Output.11	:=	QxShare159	;//	备用
ET04_Output[2].Output.12	:=	QxShare160	;//	备用
ET04_Output[2].Output.13	:=	QxShare161	;//	备用
ET04_Output[2].Output.14	:=	QxShare162	;//	备用
ET04_Output[2].Output.15	:=	QxShare163	;//	备用
END_ACTION

END_PROGRAM

// ---- POUs/002_Machine/LightsTest.TcPOU
PROGRAM LightsTest
VAR
	fbLightTestOn_TRIG: R_TRIG;
	fbLightTestOff_TRIG: F_TRIG;
 	xLightTest:BOOL;
END_VAR

LightsTest();

ACTION LightsTest:
fbLightTestOn_TRIG(CLK:=xLightTest , Q=> );
fbLightTestOff_TRIG(CLK:=xLightTest , Q=> );
IF fbLightTestOn_TRIG.Q THEN
	QxStartButtonLamp:=TRUE	;//	启动按钮指示灯
	QxStopButtonLamp:=TRUE		;//	停止按钮指示灯
  QxResetButtonLamp:=TRUE		;//	复位按钮指示灯
  QxInitButtonLamp:=TRUE		;//	初始化按钮指示灯
	QxMachineLamp1Control:=TRUE;	;//	日光灯1控制
  QxMachineLamp2Control:=TRUE;	;//	日光灯2控制
	QxRedLamp	:=TRUE;//	三色灯-红灯
	QxYellowLamp:=TRUE	;//	三色灯-黄灯
	QxGreenLamp:=TRUE	;//	三色灯-绿灯
	QxCameraLight1Trigger:=TRUE	;//	相机光源触发通道1
	QxCameraLight2Trigger:=TRUE	;//	相机光源触发通道2
	QxCameraLight3Trigger:=TRUE	;//	相机光源触发通道3
	QxCameraLight4Trigger:=TRUE	;//	相机光源触发通道4
	
	QxRedLamp_1:=TRUE	;//	三色灯-红灯
	QxYellowLamp_1:=TRUE	;//	三色灯-黄灯
  QxGreenLamp_1:=TRUE	;//	三色灯-绿灯
	QxMachineLamp3Contorl:=TRUE	;//	日光灯控制
ELSIF fbLightTestOff_TRIG.Q THEN
	QxStartButtonLamp:=FALSE	;//	启动按钮指示灯
	QxStopButtonLamp:=FALSE		;//	停止按钮指示灯
  QxResetButtonLamp:=FALSE		;//	复位按钮指示灯
  QxInitButtonLamp:=FALSE		;//	初始化按钮指示灯
	QxMachineLamp1Control:=FALSE;	;//	日光灯1控制
  QxMachineLamp2Control:=FALSE;	;//	日光灯2控制
	QxRedLamp	:=FALSE;//	三色灯-红灯
	QxYellowLamp:=FALSE	;//	三色灯-黄灯
	QxGreenLamp:=FALSE	;//	三色灯-绿灯
	QxCameraLight1Trigger:=FALSE	;//	相机光源触发通道1
	QxCameraLight2Trigger:=FALSE	;//	相机光源触发通道2
	QxCameraLight3Trigger:=FALSE	;//	相机光源触发通道3
	QxCameraLight4Trigger:=FALSE	;//	相机光源触发通道4
	
	QxRedLamp_1:=FALSE	;//	三色灯-红灯
	QxYellowLamp_1:=FALSE	;//	三色灯-黄灯
  QxGreenLamp_1:=FALSE	;//	三色灯-绿灯
	QxMachineLamp3Contorl:=FALSE	;//	日光灯控制
END_IF
END_ACTION

END_PROGRAM

// ---- POUs/003_FB/19-AxisFB/FB_AxisHome.TcPOU
FUNCTION_BLOCK FB_AxisHome
VAR_IN_OUT
	{attribute 'hide'}
	axis_name: Tc2_MC2.AXIS_REF;	
END_VAR


VAR_INPUT
  iMode : INT := 1;//驱动器模式选择；1：三菱伺服 ，2：高创伺服；3雷赛驱动
	home_exe:BOOL;
	{attribute 'hide'}
	fb_netid :Tc2_System.T_AmsNetID;
	fb_nslaveaddr  :UINT;
	nctrl1 :USINT;
	nctrl2 :USINT;

	home_method:SINT;//6098
	home_highspeed_set:REAL;//6099_01，单位rpm
	home_lowspeed_set:REAL;//6099_02，单位rpm
	home_offset_set:REAL;//607C
	numerator:REAL;//电子齿轮比分母
	denominator:REAL;//电子齿轮比分子
	//home_actpos_cal_method:UINT;//60E6
	tTimeOutSet : TIME := T#20S ;
END_VAR
VAR_OUTPUT
	home_done:BOOL;
	home_error:BOOL;
	controlword :UINT;//6040
	error_id:INT;
END_VAR
VAR_IN_OUT
	mode:SINT;//6060
END_VAR
VAR
	{attribute 'hide'}
	mc_reset:Tc2_MC2.MC_Reset;
	//fb_sdoread_6040:Tc2_EtherCAT.FB_EcCoESdoRead;
	//fb_sdowrite_6040:Tc2_EtherCAT.FB_EcCoESdoWrite;
	{attribute 'hide'}
	fb_sdoread_6041:Tc2_EtherCAT.FB_EcCoESdoRead;
	{attribute 'hide'}
	fb_sdoread_6060:Tc2_EtherCAT.FB_EcCoESdoRead;
	{attribute 'hide'}
	fb_sdowrite_6060:Tc2_EtherCAT.FB_EcCoESdoWrite;
	{attribute 'hide'}
	fb_sdoread_6098:Tc2_EtherCAT.FB_EcCoESdoRead;
	{attribute 'hide'}
	fb_sdowrite_6098:Tc2_EtherCAT.FB_EcCoESdoWrite;
	{attribute 'hide'}
	fb_sdoread_6099_01:Tc2_EtherCAT.FB_EcCoESdoRead;
	{attribute 'hide'}
	fb_sdowrite_6099_01:Tc2_EtherCAT.FB_EcCoESdoWrite;
	{attribute 'hide'}
	fb_sdoread_6099_02:Tc2_EtherCAT.FB_EcCoESdoRead;
	{attribute 'hide'}
	fb_sdowrite_6099_02:Tc2_EtherCAT.FB_EcCoESdoWrite;
	{attribute 'hide'}
	fb_sdoread_607C:Tc2_EtherCAT.FB_EcCoESdoRead;
	{attribute 'hide'}
	fb_sdowrite_607C:Tc2_EtherCAT.FB_EcCoESdoWrite;
	{attribute 'hide'}
	fb_sdoread_6091_01:Tc2_EtherCAT.FB_EcCoESdoRead;
	{attribute 'hide'}
	fb_sdoread_6091_02:Tc2_EtherCAT.FB_EcCoESdoRead;
	//fb_sdoread_60E6:Tc2_EtherCAT.FB_EcCoESdoRead;
	//fb_sdowrite_60E6:Tc2_EtherCAT.FB_EcCoESdoWrite;
	{attribute 'hide'}
	mcsetposition:MC_SetPosition;
	{attribute 'hide'}
	ton1:Tc2_Standard.TON;
	{attribute 'hide'}
	ton2:Tc2_Standard.TON;
	{attribute 'hide'}
	_tonDelay , _tonDelay1 , _tonDelay2 : Tc2_Standard.TON;
	
	increments:REAL:=8388608.0;
	exe_reset:BOOL;
	reset_done:BOOL;
	sdo_read:BOOL;
	home_start:BOOL:=FALSE;
	home_step:INT:=0;
	
	statusword :UINT;//_6041

	mode_display:SINT;//_6060
	home_method_display:SINT;//_6098
	home_highspeed:UDINT;//6099_01
	home_lowspeed:UDINT;//6099_02
	home_highspeed_display:UDINT;//_6099_01
	home_lowspeed_display:UDINT;//_6099_02
	home_offset_display:DINT;//_607C
	home_offset:DINT;//607C
	motor:UDINT:=1;//6091_01
	shaft:UDINT:=1;//6091_02
	//home_actpos_cal_method_display:UINT;//_60E6
	_iCount : int ;
END_VAR


home_highspeed:=REAL_TO_UDINT((((home_highspeed_set/numerator)*denominator)*UDINT_TO_REAL(motor))/UDINT_TO_REAL(shaft));
home_lowspeed:=REAL_TO_UDINT((((home_lowspeed_set/numerator)*denominator)*UDINT_TO_REAL(motor))/UDINT_TO_REAL(shaft));
home_offset:=REAL_TO_DINT(((((home_offset_set/numerator)*denominator)*UDINT_TO_REAL(motor))/UDINT_TO_REAL(shaft)));
mc_reset(Axis:=axis_name , Execute:=exe_reset , Done=>reset_done , Busy=> , Error=> , ErrorID=> );
ton1(IN:=NOT(ton1.Q) , PT:= T#20MS, Q=> , ET=> );
ton2(IN:= , PT:=T#500MS , Q=> , ET=> );
IF ton1.Q THEN sdo_read:=TRUE; ELSE sdo_read:=FALSE; END_IF

IF home_start=FALSE THEN 
	controlword.0:=nctrl1.0;controlword.1:=nctrl1.1;controlword.2:=nctrl1.2;controlword.3:=nctrl1.3;controlword.4:=nctrl1.4;controlword.5:=nctrl1.5;controlword.6:=nctrl1.6;controlword.7:=nctrl1.7;
    controlword.8:=nctrl2.0;controlword.9:=nctrl2.1;controlword.10:=nctrl2.2;controlword.11:=nctrl2.3;controlword.12:=nctrl2.4;controlword.13:=nctrl2.5;controlword.14:=nctrl2.6;controlword.15:=nctrl2.7;
END_IF


